// TwinCAT 3 PLC project IMD_PLC
// ProgramVersion: 3.1.4020.4
// libraries:
//   Tc2_ControllerToolbox, * (Beckhoff Automation GmbH)
//   Tc2_Database, * (Beckhoff Automation GmbH)
//   Tc2_Drive, * (Beckhoff Automation GmbH)
//   Tc2_EtherCAT, * (Beckhoff Automation GmbH)
//   Tc2_MC2, * (Beckhoff Automation GmbH)
//   Tc2_Standard, * (Beckhoff Automation GmbH)
//   Tc2_System, * (Beckhoff Automation GmbH)
//   Tc2_Utilities, * (Beckhoff Automation GmbH)
//   Tc3_Database, * (Beckhoff Automation GmbH)
//   Tc3_EventLogger, * (Beckhoff Automation GmbH)
//   Tc3_Module, * (Beckhoff Automation GmbH)
// project tree:
//   DUTs/ ST_COM_SpeedControl.TcDUT, ST_COM_IMD_SpdCntrl.TcDUT, ST_MachPar.TcDUT, ST_OEE.TcDUT, ST_PowerMeasurement.TcDUT, ST_ProdPar.TcDUT, ST_COM_SpdCntrl_IMD.TcDUT, ST_Record.TcDUT, ST_SysPar.TcDUT
//   GVLs/ GVL.TcGVL
//   / PlcTask.TcTTO, RecipeManager.TcRMO (not stored)
//   POUs/ FB_instancePath.TcPOU, HMI.TcPOU, MAIN.TcPOU, ST_Errors.TcDUT
//   POUs/InMoldDrying/BottomMold/ FB_BottomMold.TcPOU, ST_BottomMoldErrors.TcDUT, ST_BottomMoldMachPar.TcDUT, ST_BottomMoldProdPar.TcDUT, ST_BottomMoldSysPar.TcDUT
//   POUs/InMoldDrying/ FB_InMoldDrying.TcPOU, ST_IMDErrors.TcDUT, ST_IMDMachPar.TcDUT, ST_IMDProdPar.TcDUT, ST_IMDSysPar.TcDUT
//   POUs/InMoldDrying/HydrolicsMain/ FB_HydraulicsMain.TcPOU, ST_HydraulicsMainErrors.TcDUT, ST_HydraulicsMainMachPar.TcDUT
//   POUs/InMoldDrying/ProductForming/ FB_ProductForming.TcPOU, ST_FormingMoldErrors.TcDUT, ST_FormingMoldMachPar.TcDUT, ST_MachinePondErrors.TcDUT, ST_MachinePondMachPar.TcDUT, ST_ProductFormingErrors.TcDUT, ST_ProductFormingMachPar.TcDUT, ST_ProductFormingSysPar.TcDUT, ST_SpraybarErrors.TcDUT, ST_SpraybarMachPar.TcDUT
//   POUs/InMoldDrying/TopMold/ FB_TopMold.TcPOU, ST_TopMoldErrors.TcDUT, ST_TopMoldMachPar.TcDUT, ST_TopMoldProdPar.TcDUT
//   POUs/InMoldDrying/TransferMold/ FB_TransferMold.TcPOU, ST_TransferMoldErrors.TcDUT, ST_TransferMoldMachPar.TcDUT, ST_TransferMoldProdPar.TcDUT
//   POUs/ProductHandling/ FB_Gantry.TcPOU, FB_ProductHandling.TcPOU, ST_BlowOffProdPar.TcDUT, ST_GantryMachPar.TcDUT, ST_GantryProdPar.TcDUT, ST_GantryErrors.TcDUT, ST_GantrySysPar.TcDUT, ST_ProductHandlingErrors.TcDUT, ST_ProductHandlingMachPar.TcDUT, ST_ProductHandlingProdPar.TcDUT, ST_ProductHandlingSysPar.TcDUT
//   POUs/Standard/Analog/ FB_AnalogIn4_20mA.TcPOU, FB_AnalogInPT100.TcPOU, FB_AnalogOut0_10V.TcPOU, FB_AnalogOutMinus10_10V.TcPOU
//   POUs/Standard/Balluff/ FB_BalluffDevice.TcPOU, FB_BalluffPosition.TcPOU, ST_BalluffDevice.TcDUT, ST_BalluffMagnet.TcDUT
//   POUs/Standard/ FB_Blink.TcPOU, FB_EthercatDiag.TcPOU, GateRequest.TcPOU, UnixTimestamp.TcPOU
//   POUs/Standard/FIFO/ FB_CalculateMaxKO.TcPOU
//   POUs/Standard/HeatingZone/ FB_HeatingZone.TcPOU, ST_HeatingZoneErrors.TcDUT, ST_HeatingZone.TcDUT
//   POUs/Standard/HeatingZone/PID/ FB_1stOrderFilter.TcPOU, FB_PID.TcPOU, FB_PIDCtrl.TcPOU, FB_PID_CP.TcPOU, FB_PID_ROC.TcPOU, ST_PIDSettings.TcDUT
//   POUs/Standard/HydraulicCylinderAnalog/ FB_HydraulicCilinderAnalog.TcPOU, FB_HydraulicCilinderAnalog_.TcPOU, ST_HydraulicCilinderMachParAnalog.TcDUT, ST_HydraulicErrorsAnalog.TcDUT
//   POUs/Standard/Motor/ FB_Motor.TcPOU, FB_MotorSS.TcPOU, ST_MotorSSErrors.TcDUT, ST_MotorErrors.TcDUT
//   POUs/Standard/NC_Axis/ FB_NcAxis.TcPOU, ST_NcAxis_Errors.TcDUT, ST_NcAxis_Parameters_XX.TcDUT, ST_NcAxis_SysPar.TcDUT
//   POUs/Standard/HydraulicCilinder/ FB_HydraulicCilinder.TcPOU, ST_HydraulicCilinderMachPar.TcDUT, ST_HydraulicErrors.TcDUT
//   POUs/Standard/Valves/ FB_MonoValve2Fdbck.TcPOU, FB_CheckCilinder.TcPOU, FB_MonoValveNoFdbck.TcPOU, FB_BiValve2Fdbck.TcPOU, ST_CilinderErrors.TcDUT, ST_CilinderParameters.TcDUT
// real-time tasks:
//   TASK PlcTask: cycle T#10ms, priority 20, ADS port 350
//   TASK PlcTask_SpeedControl: cycle T#2ms, priority 19, ADS port 351
// motion (NC):
//   TASK NC-Task 1 SAF: cycle T#2ms, priority 4, ADS port 501
//   TASK NC-Task 1 SVB: cycle T#10ms, priority 8, ADS port 511
//   AXIS GantryA_Hor (id 1)
//     Dynamic: AccelerationMaximum=1657, DecelerationMaximum=1800, Acceleration=6750, Deceleration=6750, Jerk=50625
//     Velo: RefSearch=180, RefSync=180, SlowManual=165, FastManual=360, Fast=18000, Maximum=1800
//     OtherSettings: AllowMotionCmdToSlave=true
//     encoder EncType=8
//       EncPara: ScaleFactorNumerator=3.1607491629e-05, MaxCount=#xffffffff
//     drive DrvType=9
//       DrvPara: MaxCount=#xffffffff, DriveControlDWord=#x00030100
//         Analog: VeloReferenz=1657, VeloScale=1.02400649589962
//         TimeComp: TaskDelayCycles=1
//     controller CtrType=1
//       CtrPara: PriorControlFactor=1
//         PosDiffControl: Range=1
//         Observer: BandWidth=20
//   AXIS GantryA_Ver (id 2)
//     Dynamic: AccelerationMaximum=1000, DecelerationMaximum=1000, Acceleration=1000, Deceleration=1000, Jerk=15000
//     Velo: SlowManual=180, FastManual=450, Maximum=1000
//     OtherSettings: AllowMotionCmdToSlave=true
//     encoder EncType=8
//       EncPara: ScaleFactorNumerator=1.1444091797e-05, MaxCount=#xffffffff
//     drive DrvType=9
//       DrvPara: MaxCount=#xffffffff, DriveControlDWord=#x00030100
//         Analog: VeloReferenz=900, VeloScale=1.02400649589962
//         TimeComp: TaskDelayCycles=1
//     controller CtrType=1
//       CtrPara: PriorControlFactor=1
//         PosDiffControl: Range=0.3
//         Observer: BandWidth=20
//   AXIS GantryB_Hor (id 3)
//     Dynamic: Acceleration=5400, Deceleration=5400, Jerk=32400
//     Velo: SlowManual=165, FastManual=900, Maximum=1800
//     OtherSettings: AllowMotionCmdToSlave=true
//     encoder EncType=8
//       EncPara: ScaleFactorNumerator=3.1607491629e-05, Inverse=true, MaxCount=#xffffffff
//     drive DrvType=9
//       DrvPara: Inverse=true, MaxCount=#xffffffff, DriveControlDWord=#x00030100
//         Analog: VeloReferenz=1657, VeloScale=1.02400649589962
//         TimeComp: TaskDelayCycles=1
//     controller CtrType=1
//       CtrPara: PriorControlFactor=1
//         PosDiffControl: Range=1
//         Observer: BandWidth=20
//   AXIS GantryB_Ver (id 4)
//     Dynamic: Acceleration=3000, Deceleration=3000, Jerk=18000
//     Velo: FastManual=500, Maximum=1000
//     OtherSettings: AllowMotionCmdToSlave=true
//     encoder EncType=8
//       EncPara: ScaleFactorNumerator=1.1444091797e-05, Inverse=true, MaxCount=#xffffffff
//     drive DrvType=9
//       DrvPara: Inverse=true, MaxCount=#xffffffff, DriveControlDWord=#x00030100
//         Analog: VeloReferenz=900, VeloScale=1.02400649589962
//         TimeComp: TaskDelayCycles=1
//     controller CtrType=1
//       CtrPara: PriorControlFactor=1
//         PosDiffControl: Range=0.3
//         Observer: BandWidth=20
//   AXIS Conveyor (id 5)
//     General: UnitFlags=#x00000004
//     Dynamic: Acceleration=1368, Deceleration=1368, Jerk=8208
//     Velo: SlowManual=40, FastManual=207, Maximum=456
//     OtherSettings: AllowMotionCmdToSlave=true
//     encoder EncType=8
//       EncPara: ScaleFactorNumerator=7.780808382e-06, ModuloFactor=4620, Inverse=true, MaxCount=#xffffffff
//     drive DrvType=9
//       DrvPara: Inverse=true, MaxCount=#xffffffff, DriveControlDWord=#x00030100
//         Analog: VeloReferenz=414.74, VeloScale=1.02400649589962
//         TimeComp: TaskDelayCycles=1
//     controller CtrType=1
//       CtrPara: PriorControlFactor=1
//         Observer: BandWidth=20
//   AXIS SprayBar (id 6)
//     Dynamic: Acceleration=9780, Deceleration=9780, Jerk=58680
//     Velo: Maximum=3260
//     OtherSettings: AllowMotionCmdToSlave=true
//     encoder EncType=8
//       EncPara: ScaleFactorNumerator=5.8372727731e-05, MaxCount=#xffffffff
//     drive DrvType=9
//       DrvPara: MaxCount=#xffffffff, DriveControlDWord=#x00030100
//         Analog: VeloReferenz=2964, VeloScale=1.02400649589962
//         TimeComp: TaskDelayCycles=1
//     controller CtrType=1
//       CtrPara: PriorControlFactor=1
//         Observer: BandWidth=20
//   AXIS BottomMoldA (id 7)
//     Dynamic: AccelerationMaximum=5000, DecelerationMaximum=5000, Acceleration=1000, Deceleration=1000, Jerk=14000
//     Velo: Maximum=1250
//     OtherSettings: AllowMotionCmdToSlave=true
//     encoder EncType=8
//       EncPara: MaxCount=#xffffffff
//     drive DrvType=9
//       DrvPara: MaxCount=#xffffffff, DriveControlDWord=#x00030000
//         Analog: VeloScale=6
//         TimeComp: TaskDelayCycles=1
//     controller CtrType=1
//       CtrPara: PriorControlFactor=1
//         PosDiffControl: Enable=false, Range=15, Time=0
//         Observer: BandWidth=20
//   AXIS BottomMoldB (id 8)
//     Dynamic: Acceleration=1000, Deceleration=1000, Jerk=14000
//     OtherSettings: AllowMotionCmdToSlave=true
//     encoder EncType=8
//       EncPara: MaxCount=#xffffffff
//     drive DrvType=9
//       DrvPara: MaxCount=#xffffffff, DriveControlDWord=#x00030000
//         Analog: VeloScale=6
//         TimeComp: TaskDelayCycles=1
//     controller CtrType=1
//       CtrPara: PriorControlFactor=1
//         PosDiffControl: Enable=false
//         Observer: BandWidth=20
// I/O:
//   DEVICE Device 2 (EtherCAT) (disabled), AmsNetId 192.168.0.122.3.1
//     MCC01_600A1 (EK1100) [EK1100 EtherCAT Coupler (2A E-Bus)]
//       600A3 (EL9210) [EL9210 Power Supplier with LED (24V, Fuse, Diagnostics)]
//       600A4_TwinsafeController (EL6900) [EL6900, TwinSAFE PLC]
//       600A5 (EL2904) [EL2904, 4 Ch. Safety Output 24V, 0.5A, TwinSAFE]
//         modules: Module 1 (FSOES), Module 2 (DO)
//       600A6 (EL2904) [EL2904, 4 Ch. Safety Output 24V, 0.5A, TwinSAFE]
//         modules: Module 1 (FSOES), Module 2 (DO)
//       600A7 (EL2904) [EL2904, 4 Ch. Safety Output 24V, 0.5A, TwinSAFE]
//         modules: Module 1 (FSOES), Module 2 (DO)
//       600A8 (EL2904) [EL2904, 4 Ch. Safety Output 24V, 0.5A, TwinSAFE]
//         modules: Module 1 (FSOES), Module 2 (DO)
//       600A9 (EL9410) [EL9410 E-Bus Power Supplier  (Diagnostics)]
//       600A10 (EL2904) [EL2904, 4 Ch. Safety Output 24V, 0.5A, TwinSAFE]
//         modules: Module 1 (FSOES), Module 2 (DO)
//       600A11 (EL2904) [EL2904, 4 Ch. Safety Output 24V, 0.5A, TwinSAFE]
//         modules: Module 1 (FSOES), Module 2 (DO)
//       600A12 (EL2904) [EL2904, 4 Ch. Safety Output 24V, 0.5A, TwinSAFE]
//         modules: Module 1 (FSOES), Module 2 (DO)
//       600A13 (EL2904) [EL2904, 4 Ch. Safety Output 24V, 0.5A, TwinSAFE]
//         modules: Module 1 (FSOES), Module 2 (DO)
//       600A14 (EL2904) [EL2904, 4 Ch. Safety Output 24V, 0.5A, TwinSAFE]
//         modules: Module 1 (FSOES), Module 2 (DO)
//       600A15 (EL9210) [EL9210 Power Supplier with LED (24V, Fuse, Diagnostics)]
//       600A16 (EL1809) [EL1809 16Ch. Dig. Input 24V, 3ms]
//       600A17 (EL1809) [EL1809 16Ch. Dig. Input 24V, 3ms]
//       600A18 (EL1809) [EL1809 16Ch. Dig. Input 24V, 3ms]
//       600A19 (EL1809) [EL1809 16Ch. Dig. Input 24V, 3ms]
//       600A20 (EL1809) [EL1809 16Ch. Dig. Input 24V, 3ms]
//       600A21 (EL1809) [EL1809 16Ch. Dig. Input 24V, 3ms]
//       600A22 (EL9410) [EL9410 E-Bus Power Supplier  (Diagnostics)]
//       600A23 (EL2809) [EL2809 16Ch. Dig. Output 24V, 0.5A]
//       600A24 (EL2809) [EL2809 16Ch. Dig. Output 24V, 0.5A]
//       600A25 (EL2809) [EL2809 16Ch. Dig. Output 24V, 0.5A]
//       600A26 (EL2809) [EL2809 16Ch. Dig. Output 24V, 0.5A]
//       600A27 (EL2809) [EL2809 16Ch. Dig. Output 24V, 0.5A]
//       600A28 (EL9011) [EL9011 End Terminal]
//     MCC01_2_610A1 (EK1100) [EK1100 EtherCAT Coupler (2A E-Bus)]
//       610A1.1 (EL1809) [EL1809 16Ch. Dig. Input 24V, 3ms]
//       610A1.2 (EL2809) [EL2809 16Ch. Dig. Output 24V, 0.5A]
//       610A2 (EK1122) [EK1122 2 port EtherCAT junction]
//         Drive Gantry A (AX5203-0000-0203) [AX5203-0000-0203 EtherCAT Drive (SoE, 2 Ch.)]
//           GantryA (AX5805) [AX5805 (Safety Drive Option)]
//             modules: Module 1 (Safety Process Data, 2 axis), Module 2 (Standard Process Data, 2 axis)
//           Term 145 (EL9011) [EL9011 End Terminal]
//         Drive Gantry B (AX5203-0000-0203) [AX5203-0000-0203 EtherCAT Drive (SoE, 2 Ch.)]
//           GantryB (AX5805) [AX5805 (Safety Drive Option)]
//             modules: Module 1 (Safety Process Data, 2 axis), Module 2 (Standard Process Data, 2 axis)
//           Term 146 (EL9011) [EL9011 End Terminal]
//         Drive A-Belt / B-Spraybar (AX5201-0000-0203) [AX5201-0000-0203 EtherCAT Drive (SoE, 2 Ch.)]
//           SprayBar_Belt (AX5805) [AX5805 (Safety Drive Option)]
//             modules: Module 1 (Safety Process Data, 2 axis), Module 2 (Standard Process Data, 2 axis)
//           Term 147 (EL9011) [EL9011 End Terminal]
//         EJBox (EP9128-0021) [EP9128-0021 8x EtherCAT junction]
//           RIO_600A1 (EK1100) [EK1100 EtherCAT Coupler (2A E-Bus)]
//             RIO_600A2 (EL1804) [EL1804 4Ch. Dig. Input 24V, 3ms]
//             RIO_600A3 (EL1804) [EL1804 4Ch. Dig. Input 24V, 3ms]
//             RIO_600A4 (EL1804) [EL1804 4Ch. Dig. Input 24V, 3ms]
//             RIO_600A5 (EL1804) [EL1804 4Ch. Dig. Input 24V, 3ms]
//             RIO_600A6 (EL9210) [EL9210 Power Supplier with LED (24V, Fuse, Diagnostics)]
//             RIO_600A7 (EL2808) [EL2808 8Ch. Dig. Output 24V, 0.5A]
//             RIO_600A8 (EL2808) [EL2808 8Ch. Dig. Output 24V, 0.5A]
//             RIO_600A9 (EL2808) [EL2808 8Ch. Dig. Output 24V, 0.5A]
//             RIO_600A10 (EL9210) [EL9210 Power Supplier with LED (24V, Fuse, Diagnostics)]
//             RIO_600A11 (EL1904) [EL1904, 4 Ch. Safety Input 24V, TwinSAFE]
//               modules: Module 1 (FSOES)
//             RIO_600A12 (EL1904) [EL1904, 4 Ch. Safety Input 24V, TwinSAFE]
//               modules: Module 1 (FSOES)
//             RIO_600A13 (EL1904) [EL1904, 4 Ch. Safety Input 24V, TwinSAFE]
//               modules: Module 1 (FSOES)
//             RIO_600A14 (EL9410) [EL9410 E-Bus Power Supplier  (Diagnostics)]
//             RIO_600A15 (EL9210) [EL9210 Power Supplier with LED (24V, Fuse, Diagnostics)]
//             RIO_600A16 (EL1904) [EL1904, 4 Ch. Safety Input 24V, TwinSAFE]
//               modules: Module 1 (FSOES)
//             RIO_600A17 (EL1904) [EL1904, 4 Ch. Safety Input 24V, TwinSAFE]
//               modules: Module 1 (FSOES)
//             RIO_600A18 (EL9185) [EL9185 Potential Connection, 4 x 24-230V]
//             RIO_600A19 (EL9185) [EL9185 Potential Connection, 4 x 24-230V]
//             RIO_600A20 (EL1904) [EL1904, 4 Ch. Safety Input 24V, TwinSAFE]
//               modules: Module 1 (FSOES)
//             RIO_600A21 (EL1904) [EL1904, 4 Ch. Safety Input 24V, TwinSAFE]
//               modules: Module 1 (FSOES)
//             RIO_600A22 (EL1904) [EL1904, 4 Ch. Safety Input 24V, TwinSAFE]
//               modules: Module 1 (FSOES)
//             RIO_600A23 (EL1904) [EL1904, 4 Ch. Safety Input 24V, TwinSAFE]
//               modules: Module 1 (FSOES)
//             RIO_600A24 (EL1904) [EL1904, 4 Ch. Safety Input 24V, TwinSAFE]
//               modules: Module 1 (FSOES)
//             RIO_600A25 (EL1904) [EL1904, 4 Ch. Safety Input 24V, TwinSAFE]
//               modules: Module 1 (FSOES)
//             RIO_600A26 (EL1904) [EL1904, 4 Ch. Safety Input 24V, TwinSAFE]
//               modules: Module 1 (FSOES)
//             RIO_600A27 (EL9185) [EL9185 Potential Connection, 4 x 24-230V]
//             RIO_600A28 (EL9185) [EL9185 Potential Connection, 4 x 24-230V]
//             RIO_600A29 (EL9185) [EL9185 Potential Connection, 4 x 24-230V]
//             RIO_600A30 (EL9185) [EL9185 Potential Connection, 4 x 24-230V]
//             RIO_600A31 (EL3052) [EL3052 2Ch. Ana. Input 4-20mA]
//             RIO_600A32 (EL9011) [EL9011 End Terminal]
//           EPP_SensorSpeedControl (EPP1322-0001) [EPP1322-0001 3 port EtherCAT P gateway]
//             Box SpeedControl (EPP6228-0022) [EPP6228 (IO Link Master)]
//               modules: Module 1 (DeviceState Inputs Device), Module 2 (DeviceState Inputs), Module 3 (IO-Link Slave), Module 4 (empty), Module 5 (empty), Module 6 (empty), Module 7 (empty), Module 8 (empty), Module 9 (empty), Module 10 (empty), Module 11 (Digital Inputs)
//           TopMoldA (BTL7 EtherCAT) [BTL7 EtherCAT Modular]
//             modules: Module 1 (Position, speed, state, CAM and workarea), Module 17 (Error register and temperature), Module 18 (1 Magnet)
//           TransferMold (BTL7 EtherCAT) [BTL7 EtherCAT Modular]
//             modules: Module 1 (Position, speed, state, CAM and workarea), Module 17 (Error register and temperature), Module 18 (1 Magnet)
//           TopMoldB (BTL7 EtherCAT) [BTL7 EtherCAT Modular]
//             modules: Module 1 (Position, speed, state, CAM and workarea), Module 17 (Error register and temperature), Module 18 (1 Magnet)
//           BottomMoldHorizontal (BTL7 EtherCAT) [BTL7 EtherCAT Modular]
//             modules: Module 1 (Position, speed, state, CAM and workarea), Module 2 (Position, speed, state, CAM and workarea), Module 17 (Error register and temperature), Module 18 (2 Magnets)
//           MachinePond (BTL7 EtherCAT) [BTL7 EtherCAT Modular]
//             modules: Module 1 (Position, speed, state, CAM and workarea), Module 17 (Error register and temperature), Module 18 (1 Magnet)
//           JB_ (EP9128-1021) [EP9128-1021 8x EtherCAT junction - Dev A]
//             Box B (EP2008-0001) [EP2008-0001 8 Ch. Dig. Output 24V, 0,5A, M8]
//             Box Y1 [EP3174-0002 4Ch. Ana. Input +/-10V, 0-10V, 0/4-20mA configurable]
//             Box Y2 (EP3174-0002) [EP3174-0002 4Ch. Ana. Input +/-10V, 0-10V, 0/4-20mA configurable]
//             Box D (EP2028-0001) [EP2028-0001 8 Ch. Dig. Output 24V, 2A, M8]
//             Box A (EP2028-0001) [EP2028-0001 8 Ch. Dig. Output 24V, 2A, M8]
//             Box X (EP3174-0002) [EP3174-0002 4Ch. Ana. Input +/-10V, 0-10V, 0/4-20mA configurable]
//             Box C (EP2008-0001) [EP2008-0001 8 Ch. Dig. Output 24V, 0,5A, M8]
//             Box J (EP2008-0001) [EP2008-0001 8 Ch. Dig. Output 24V, 0,5A, M8]
//             Box AA (EP1008-0001) [EP1008-0001 8 Ch. Dig. Input 24V, 3ms, M8]
//             Box EF (EP2308-0001) [EP2308-0001 4 Ch. Dig. In, 3ms, 4 Ch. Dig. Out 24V, 0,5A, M8]
//             Box K (EP2008-0001) [EP2008-0001 8 Ch. Dig. Output 24V, 0,5A, M8]
//             Box L (EP1008-0001) [EP1008-0001 8 Ch. Dig. Input 24V, 3ms, M8]
//           JB_BottomMoldB_GantryA (EP9128-2021) [EP9128-2021 8x EtherCAT junction - Dev B]
//             Box HI (EP2308-0001) [EP2308-0001 4 Ch. Dig. In, 3ms, 4 Ch. Dig. Out 24V, 0,5A, M8]
//             Box M (EP2008-0001) [EP2008-0001 8 Ch. Dig. Output 24V, 0,5A, M8]
//             Box N (EP1008-0001) [EP1008-0001 8 Ch. Dig. Input 24V, 3ms, M8]
//             Box O (EP1008-0001) [EP1008-0001 8 Ch. Dig. Input 24V, 3ms, M8]
//             Box P (EP1008-0001) [EP1008-0001 8 Ch. Dig. Input 24V, 3ms, M8]
//             Box R (EP1008-0001) [EP1008-0001 8 Ch. Dig. Input 24V, 3ms, M8]
//             Box Q1 (EP2008-0001) [EP2008-0001 8 Ch. Dig. Output 24V, 0,5A, M8]
//             Box Q2 (EP2008-0001) [EP2008-0001 8 Ch. Dig. Output 24V, 0,5A, M8]
//         Box S (gantry B) (EP1008-0001) [EP1008-0001 8 Ch. Dig. Input 24V, 3ms, M8]
//         Box T (gantry B) (EP1008-0001) [EP1008-0001 8 Ch. Dig. Input 24V, 3ms, M8]
//         Box V (gantry B) (EP1008-0001) [EP1008-0001 8 Ch. Dig. Input 24V, 3ms, M8]
//         Box U1 (gantry B) (EP2008-0001) [EP2008-0001 8 Ch. Dig. Output 24V, 0,5A, M8]
//         Box U2 (gantry B) (EP2008-0001) [EP2008-0001 8 Ch. Dig. Output 24V, 0,5A, M8]
//       610A3 (EL9210) [EL9210 Power Supplier with LED (24V, Fuse, Diagnostics)]
//       610A4 (EL3403) [EL3403 3Ch. Power Measuring]
//       610A5 (EL3202) [EL3202 2Ch. Ana. Input PT100 (RTD)]
//       610A6 (EL3202) [EL3202 2Ch. Ana. Input PT100 (RTD)]
//       610A7 (EL3202) [EL3202 2Ch. Ana. Input PT100 (RTD)]
//       610A8 (EL3202) [EL3202 2Ch. Ana. Input PT100 (RTD)]
//       610A9 (EL3202) [EL3202 2Ch. Ana. Input PT100 (RTD)]
//       610A10 (EL3202) [EL3202 2Ch. Ana. Input PT100 (RTD)]
//       610A11 (EL3202) [EL3202 2Ch. Ana. Input PT100 (RTD)]
//       610A12 (EL9410) [EL9410 E-Bus Power Supplier  (Diagnostics)]
//       610A13 (EL3202) [EL3202 2Ch. Ana. Input PT100 (RTD)]
//       610A14 (EL3202) [EL3202 2Ch. Ana. Input PT100 (RTD)]
//       610A15 (EL3202) [EL3202 2Ch. Ana. Input PT100 (RTD)]
//       610A16 (EL3202) [EL3202 2Ch. Ana. Input PT100 (RTD)]
//       610A17 (EL3202) [EL3202 2Ch. Ana. Input PT100 (RTD)]
//       610A18 (EL9210) [EL9210 Power Supplier with LED (24V, Fuse, Diagnostics)]
//       610A19 (EL4002) [EL4002 2Ch. Ana. Output 0-10V, 12bit]
//       610A19.1 (EL3022) [EL3022 2Ch. Ana. Input 4-20mA DIFF]
//       610A20 (EL1904) [EL1904, 4 Ch. Safety Input 24V, TwinSAFE]
//         modules: Module 1 (FSOES)
//       610A21 (EL1904) [EL1904, 4 Ch. Safety Input 24V, TwinSAFE]
//         modules: Module 1 (FSOES)
//       610A22 (EL9011) [EL9011 End Terminal]
//     MCC02_600A1 (EK1100) [EK1100 EtherCAT Coupler (2A E-Bus)]
//       MCC02_600A2 (EL1904) [EL1904, 4 Ch. Safety Input 24V, TwinSAFE]
//         modules: Module 1 (FSOES)
//       MCC02_600A3 (EL1904) [EL1904, 4 Ch. Safety Input 24V, TwinSAFE]
//         modules: Module 1 (FSOES)
//       MCC02_600A4 (EL2904) [EL2904, 4 Ch. Safety Output 24V, 0.5A, TwinSAFE]
//         modules: Module 1 (FSOES), Module 2 (DO)
//       MCC02_600A5 (EL1809) [EL1809 16Ch. Dig. Input 24V, 3ms]
//       MCC02_600A6 (EL1809) [EL1809 16Ch. Dig. Input 24V, 3ms]
//       MCC02_600A7 (EL1809) [EL1809 16Ch. Dig. Input 24V, 3ms]
//       MCC02_600A8 (EL2809) [EL2809 16Ch. Dig. Output 24V, 0.5A]
//       MCC02_600A9 (EL4134) [EL4134 4Ch. Ana. Output -10/+10V, 16bit]
//       MCC02_600A10 (EL9011) [EL9011 End Terminal]
//     BottomMoldA (IndraDrive MPB20/21) [IndraDrive MPB20/21]
//     BottomMoldB (IndraDrive MPB20/21) [IndraDrive MPB20/21]
// variable links:
//   Device 2 (EtherCAT) <-> Device 2 (EtherCAT)/MCC01_2_610A1 (EK1100)/610A2 (EK1122)/Drive A-Belt / B-Spraybar (AX5201-0000-0203)/SprayBar_Belt (AX5805)
//     MCC01_600A1 (EK1100)/600A4_TwinsafeController (EL6900)/ConnectionInputs/Message_215 TxPDO <-> Module 1 (Safety Process Data, 2 axis)/Outputs (Controlword)/FSOE
//   Device 2 (EtherCAT) <-> Device 2 (EtherCAT)/MCC01_2_610A1 (EK1100)/610A2 (EK1122)/Drive Gantry A (AX5203-0000-0203)/GantryA (AX5805)
//     MCC01_600A1 (EK1100)/600A4_TwinsafeController (EL6900)/ConnectionOutputs/Message_213 RxPDO <-> Module 1 (Safety Process Data, 2 axis)/Inputs (Statusword)/FSOE
//   Device 2 (EtherCAT) <-> Device 2 (EtherCAT)/MCC01_2_610A1 (EK1100)/610A2 (EK1122)/Drive Gantry B (AX5203-0000-0203)/GantryB (AX5805)
//     MCC01_600A1 (EK1100)/600A4_TwinsafeController (EL6900)/ConnectionInputs/Message_214 TxPDO <-> Module 1 (Safety Process Data, 2 axis)/Outputs (Controlword)/FSOE
//   Device 2 (EtherCAT) <-> Device 2 (EtherCAT)/MCC01_2_610A1 (EK1100)/610A2 (EK1122)/EJBox (EP9128-0021)/RIO_600A1 (EK1100)/RIO_600A11 (EL1904)
//     MCC01_600A1 (EK1100)/600A4_TwinsafeController (EL6900)/ConnectionOutputs/Message_128 RxPDO <-> Module 1 (FSOES)/TxPDO/FSOE
//   Device 2 (EtherCAT) <-> Device 2 (EtherCAT)/MCC01_2_610A1 (EK1100)/610A2 (EK1122)/EJBox (EP9128-0021)/RIO_600A1 (EK1100)/RIO_600A13 (EL1904)
//     MCC01_600A1 (EK1100)/600A4_TwinsafeController (EL6900)/ConnectionOutputs/Message_130 RxPDO <-> Module 1 (FSOES)/TxPDO/FSOE
//   Device 2 (EtherCAT) <-> Device 2 (EtherCAT)/MCC01_2_610A1 (EK1100)/610A2 (EK1122)/EJBox (EP9128-0021)/RIO_600A1 (EK1100)/RIO_600A17 (EL1904)
//     MCC01_600A1 (EK1100)/600A4_TwinsafeController (EL6900)/ConnectionOutputs/Message_132 RxPDO <-> Module 1 (FSOES)/TxPDO/FSOE
//   Device 2 (EtherCAT) <-> Device 2 (EtherCAT)/MCC01_2_610A1 (EK1100)/610A2 (EK1122)/EJBox (EP9128-0021)/RIO_600A1 (EK1100)/RIO_600A20 (EL1904)
//     MCC01_600A1 (EK1100)/600A4_TwinsafeController (EL6900)/ConnectionInputs/Message_133 TxPDO <-> Module 1 (FSOES)/RxPDO/FSOE
//   Device 2 (EtherCAT) <-> Device 2 (EtherCAT)/MCC01_2_610A1 (EK1100)/610A2 (EK1122)/EJBox (EP9128-0021)/RIO_600A1 (EK1100)/RIO_600A21 (EL1904)
//     MCC01_600A1 (EK1100)/600A4_TwinsafeController (EL6900)/ConnectionInputs/Message_134 TxPDO <-> Module 1 (FSOES)/RxPDO/FSOE
//     MCC01_600A1 (EK1100)/600A4_TwinsafeController (EL6900)/ConnectionOutputs/Message_134 RxPDO <-> Module 1 (FSOES)/TxPDO/FSOE
//   Device 2 (EtherCAT) <-> Device 2 (EtherCAT)/MCC01_2_610A1 (EK1100)/610A2 (EK1122)/EJBox (EP9128-0021)/RIO_600A1 (EK1100)/RIO_600A22 (EL1904)
//     MCC01_600A1 (EK1100)/600A4_TwinsafeController (EL6900)/ConnectionInputs/Message_135 TxPDO <-> Module 1 (FSOES)/RxPDO/FSOE
//   Device 2 (EtherCAT) <-> Device 2 (EtherCAT)/MCC01_2_610A1 (EK1100)/610A2 (EK1122)/EJBox (EP9128-0021)/RIO_600A1 (EK1100)/RIO_600A23 (EL1904)
//     MCC01_600A1 (EK1100)/600A4_TwinsafeController (EL6900)/ConnectionInputs/Message_136 TxPDO <-> Module 1 (FSOES)/RxPDO/FSOE
//   Device 2 (EtherCAT) <-> Device 2 (EtherCAT)/MCC01_2_610A1 (EK1100)/610A2 (EK1122)/EJBox (EP9128-0021)/RIO_600A1 (EK1100)/RIO_600A24 (EL1904)
//     MCC01_600A1 (EK1100)/600A4_TwinsafeController (EL6900)/ConnectionInputs/Message_137 TxPDO <-> Module 1 (FSOES)/RxPDO/FSOE
//   Device 2 (EtherCAT) <-> Device 2 (EtherCAT)/MCC01_2_610A1 (EK1100)/610A2 (EK1122)/EJBox (EP9128-0021)/RIO_600A1 (EK1100)/RIO_600A25 (EL1904)
//     MCC01_600A1 (EK1100)/600A4_TwinsafeController (EL6900)/ConnectionInputs/Message_138 TxPDO <-> Module 1 (FSOES)/RxPDO/FSOE
//   Device 2 (EtherCAT) <-> Device 2 (EtherCAT)/MCC01_2_610A1 (EK1100)/610A2 (EK1122)/EJBox (EP9128-0021)/RIO_600A1 (EK1100)/RIO_600A26 (EL1904)
//     MCC01_600A1 (EK1100)/600A4_TwinsafeController (EL6900)/ConnectionInputs/Message_139 TxPDO <-> Module 1 (FSOES)/RxPDO/FSOE
//   Device 2 (EtherCAT) <-> Device 2 (EtherCAT)/MCC01_2_610A1 (EK1100)/610A20 (EL1904)
//     MCC01_600A1 (EK1100)/600A4_TwinsafeController (EL6900)/ConnectionOutputs/Message_140 RxPDO <-> Module 1 (FSOES)/TxPDO/FSOE
//   Device 2 (EtherCAT) <-> Device 2 (EtherCAT)/MCC01_600A1 (EK1100)/600A10 (EL2904)
//     MCC01_600A1 (EK1100)/600A4_TwinsafeController (EL6900)/ConnectionOutputs/Message_120 RxPDO <-> Module 1 (FSOES)/TxPDO/FSOE
//   Device 2 (EtherCAT) <-> Device 2 (EtherCAT)/MCC01_600A1 (EK1100)/600A11 (EL2904)
//     MCC01_600A1 (EK1100)/600A4_TwinsafeController (EL6900)/ConnectionInputs/Message_121 TxPDO <-> Module 1 (FSOES)/RxPDO/FSOE
//   Device 2 (EtherCAT) <-> Device 2 (EtherCAT)/MCC01_600A1 (EK1100)/600A13 (EL2904)
//     MCC01_600A1 (EK1100)/600A4_TwinsafeController (EL6900)/ConnectionInputs/Message_123 TxPDO <-> Module 1 (FSOES)/RxPDO/FSOE
//     MCC01_600A1 (EK1100)/600A4_TwinsafeController (EL6900)/ConnectionOutputs/Message_123 RxPDO <-> Module 1 (FSOES)/TxPDO/FSOE
//   Device 2 (EtherCAT) <-> Device 2 (EtherCAT)/MCC01_600A1 (EK1100)/600A16 (EL1809)
//     MCC01_600A1 (EK1100)/600A4_TwinsafeController (EL6900)/StandardOutputs/Standard In Var 142 <-> Channel 2/HydroPumpFB
//     MCC01_600A1 (EK1100)/600A4_TwinsafeController (EL6900)/StandardOutputs/Standard In Var 143 <-> Channel 5/PulpPumpFB
//   Device 2 (EtherCAT) <-> Device 2 (EtherCAT)/MCC01_600A1 (EK1100)/600A18 (EL1809)
//     MCC01_600A1 (EK1100)/600A4_TwinsafeController (EL6900)/StandardOutputs/Standard In Var 196 <-> Channel 16/Input
//   Device 2 (EtherCAT) <-> Device 2 (EtherCAT)/MCC01_600A1 (EK1100)/600A21 (EL1809)
//     MCC01_600A1 (EK1100)/600A4_TwinsafeController (EL6900)/StandardOutputs/Standard In Var 189 <-> Channel 2/Chan2
//     MCC01_600A1 (EK1100)/600A4_TwinsafeController (EL6900)/StandardOutputs/Standard In Var 190 <-> Channel 1/Chan1
//     MCC01_600A1 (EK1100)/600A4_TwinsafeController (EL6900)/StandardOutputs/Standard In Var 191 <-> Channel 3/Chan3
//     MCC01_600A1 (EK1100)/600A4_TwinsafeController (EL6900)/StandardOutputs/Standard In Var 192 <-> Channel 5/Chan5
//   Device 2 (EtherCAT) <-> Device 2 (EtherCAT)/MCC01_600A1 (EK1100)/600A4_TwinsafeController (EL6900)
//     MCC01_2_610A1 (EK1100)/610A2 (EK1122)/Drive A-Belt / B-Spraybar (AX5201-0000-0203)/SprayBar_Belt (AX5805)/Module 1 (Safety Process Data, 2 axis)/Inputs (Statusword)/FSOE <-> ConnectionOutputs/Message_215 RxPDO
//     MCC01_2_610A1 (EK1100)/610A2 (EK1122)/Drive Gantry A (AX5203-0000-0203)/GantryA (AX5805)/Module 1 (Safety Process Data, 2 axis)/Outputs (Controlword)/FSOE <-> ConnectionInputs/Message_213 TxPDO
//     MCC01_2_610A1 (EK1100)/610A2 (EK1122)/Drive Gantry B (AX5203-0000-0203)/GantryB (AX5805)/Module 1 (Safety Process Data, 2 axis)/Inputs (Statusword)/FSOE <-> ConnectionOutputs/Message_214 RxPDO
//     MCC01_2_610A1 (EK1100)/610A2 (EK1122)/EJBox (EP9128-0021)/RIO_600A1 (EK1100)/RIO_600A11 (EL1904)/Module 1 (FSOES)/RxPDO/FSOE <-> ConnectionInputs/Message_128 TxPDO
//     MCC01_2_610A1 (EK1100)/610A2 (EK1122)/EJBox (EP9128-0021)/RIO_600A1 (EK1100)/RIO_600A12 (EL1904)/Module 1 (FSOES)/RxPDO/FSOE <-> ConnectionInputs/Message_129 TxPDO
//     MCC01_2_610A1 (EK1100)/610A2 (EK1122)/EJBox (EP9128-0021)/RIO_600A1 (EK1100)/RIO_600A13 (EL1904)/Module 1 (FSOES)/RxPDO/FSOE <-> ConnectionInputs/Message_130 TxPDO
//     MCC01_2_610A1 (EK1100)/610A2 (EK1122)/EJBox (EP9128-0021)/RIO_600A1 (EK1100)/RIO_600A16 (EL1904)/Module 1 (FSOES)/RxPDO/FSOE <-> ConnectionInputs/Message_131 TxPDO
//     MCC01_2_610A1 (EK1100)/610A2 (EK1122)/EJBox (EP9128-0021)/RIO_600A1 (EK1100)/RIO_600A17 (EL1904)/Module 1 (FSOES)/RxPDO/FSOE <-> ConnectionInputs/Message_132 TxPDO
//     MCC01_2_610A1 (EK1100)/610A2 (EK1122)/EJBox (EP9128-0021)/RIO_600A1 (EK1100)/RIO_600A12 (EL1904)/Module 1 (FSOES)/TxPDO/FSOE <-> ConnectionOutputs/Message_129 RxPDO
//     MCC01_2_610A1 (EK1100)/610A2 (EK1122)/EJBox (EP9128-0021)/RIO_600A1 (EK1100)/RIO_600A16 (EL1904)/Module 1 (FSOES)/TxPDO/FSOE <-> ConnectionOutputs/Message_131 RxPDO
//     MCC01_2_610A1 (EK1100)/610A2 (EK1122)/EJBox (EP9128-0021)/RIO_600A1 (EK1100)/RIO_600A20 (EL1904)/Module 1 (FSOES)/TxPDO/FSOE <-> ConnectionOutputs/Message_133 RxPDO
//     MCC01_2_610A1 (EK1100)/610A2 (EK1122)/EJBox (EP9128-0021)/RIO_600A1 (EK1100)/RIO_600A22 (EL1904)/Module 1 (FSOES)/TxPDO/FSOE <-> ConnectionOutputs/Message_135 RxPDO
//     MCC01_2_610A1 (EK1100)/610A2 (EK1122)/EJBox (EP9128-0021)/RIO_600A1 (EK1100)/RIO_600A23 (EL1904)/Module 1 (FSOES)/TxPDO/FSOE <-> ConnectionOutputs/Message_136 RxPDO
//     MCC01_2_610A1 (EK1100)/610A2 (EK1122)/EJBox (EP9128-0021)/RIO_600A1 (EK1100)/RIO_600A24 (EL1904)/Module 1 (FSOES)/TxPDO/FSOE <-> ConnectionOutputs/Message_137 RxPDO
//     MCC01_2_610A1 (EK1100)/610A2 (EK1122)/EJBox (EP9128-0021)/RIO_600A1 (EK1100)/RIO_600A25 (EL1904)/Module 1 (FSOES)/TxPDO/FSOE <-> ConnectionOutputs/Message_138 RxPDO
//     MCC01_2_610A1 (EK1100)/610A2 (EK1122)/EJBox (EP9128-0021)/RIO_600A1 (EK1100)/RIO_600A26 (EL1904)/Module 1 (FSOES)/TxPDO/FSOE <-> ConnectionOutputs/Message_139 RxPDO
//     MCC01_2_610A1 (EK1100)/610A20 (EL1904)/Module 1 (FSOES)/RxPDO/FSOE <-> ConnectionInputs/Message_140 TxPDO
//     MCC01_2_610A1 (EK1100)/610A21 (EL1904)/Module 1 (FSOES)/RxPDO/FSOE <-> ConnectionInputs/Message_141 TxPDO
//     MCC01_2_610A1 (EK1100)/610A21 (EL1904)/Module 1 (FSOES)/TxPDO/FSOE <-> ConnectionOutputs/Message_141 RxPDO
//     MCC01_600A1 (EK1100)/600A10 (EL2904)/Module 1 (FSOES)/RxPDO/FSOE <-> ConnectionInputs/Message_120 TxPDO
//     MCC01_600A1 (EK1100)/600A12 (EL2904)/Module 1 (FSOES)/RxPDO/FSOE <-> ConnectionInputs/Message_122 TxPDO
//     MCC01_600A1 (EK1100)/600A14 (EL2904)/Module 1 (FSOES)/RxPDO/FSOE <-> ConnectionInputs/Message_124 TxPDO
//     MCC01_600A1 (EK1100)/600A5 (EL2904)/Module 1 (FSOES)/RxPDO/FSOE <-> ConnectionInputs/Message_116 TxPDO
//     MCC01_600A1 (EK1100)/600A7 (EL2904)/Module 1 (FSOES)/RxPDO/FSOE <-> ConnectionInputs/Message_118 TxPDO
//     MCC01_600A1 (EK1100)/600A8 (EL2904)/Module 1 (FSOES)/RxPDO/FSOE <-> ConnectionInputs/Message_119 TxPDO
//     MCC01_600A1 (EK1100)/600A11 (EL2904)/Module 1 (FSOES)/TxPDO/FSOE <-> ConnectionOutputs/Message_121 RxPDO
//     MCC01_600A1 (EK1100)/600A12 (EL2904)/Module 1 (FSOES)/TxPDO/FSOE <-> ConnectionOutputs/Message_122 RxPDO
//     MCC01_600A1 (EK1100)/600A14 (EL2904)/Module 1 (FSOES)/TxPDO/FSOE <-> ConnectionOutputs/Message_124 RxPDO
//     MCC01_600A1 (EK1100)/600A21 (EL1809)/Channel 4/Chan4 <-> StandardOutputs/Standard In Var 188
//     MCC02_600A1 (EK1100)/MCC02_600A3 (EL1904)/Module 1 (FSOES)/RxPDO/FSOE <-> ConnectionInputs/Message_223 TxPDO
//     MCC02_600A1 (EK1100)/MCC02_600A4 (EL2904)/Module 1 (FSOES)/RxPDO/FSOE <-> ConnectionInputs/Message_218 TxPDO
//     MCC02_600A1 (EK1100)/MCC02_600A6 (EL1809)/Channel 13/Input <-> StandardOutputs/Standard In Var 220
//   Device 2 (EtherCAT) <-> Device 2 (EtherCAT)/MCC01_600A1 (EK1100)/600A5 (EL2904)
//     MCC01_600A1 (EK1100)/600A4_TwinsafeController (EL6900)/ConnectionOutputs/Message_116 RxPDO <-> Module 1 (FSOES)/TxPDO/FSOE
//   Device 2 (EtherCAT) <-> Device 2 (EtherCAT)/MCC01_600A1 (EK1100)/600A6 (EL2904)
//     MCC01_600A1 (EK1100)/600A4_TwinsafeController (EL6900)/ConnectionInputs/Message_117 TxPDO <-> Module 1 (FSOES)/RxPDO/FSOE
//     MCC01_600A1 (EK1100)/600A4_TwinsafeController (EL6900)/ConnectionOutputs/Message_117 RxPDO <-> Module 1 (FSOES)/TxPDO/FSOE
//   Device 2 (EtherCAT) <-> Device 2 (EtherCAT)/MCC01_600A1 (EK1100)/600A7 (EL2904)
//     MCC01_600A1 (EK1100)/600A4_TwinsafeController (EL6900)/ConnectionOutputs/Message_118 RxPDO <-> Module 1 (FSOES)/TxPDO/FSOE
//   Device 2 (EtherCAT) <-> Device 2 (EtherCAT)/MCC01_600A1 (EK1100)/600A8 (EL2904)
//     MCC01_600A1 (EK1100)/600A4_TwinsafeController (EL6900)/ConnectionOutputs/Message_119 RxPDO <-> Module 1 (FSOES)/TxPDO/FSOE
//   Device 2 (EtherCAT) <-> Device 2 (EtherCAT)/MCC02_600A1 (EK1100)/MCC02_600A2 (EL1904)
//     MCC01_600A1 (EK1100)/600A4_TwinsafeController (EL6900)/ConnectionInputs/Message_222 TxPDO <-> Module 1 (FSOES)/RxPDO/FSOE
//     MCC01_600A1 (EK1100)/600A4_TwinsafeController (EL6900)/ConnectionOutputs/Message_222 RxPDO <-> Module 1 (FSOES)/TxPDO/FSOE
//   Device 2 (EtherCAT) <-> Device 2 (EtherCAT)/MCC02_600A1 (EK1100)/MCC02_600A3 (EL1904)
//     MCC01_600A1 (EK1100)/600A4_TwinsafeController (EL6900)/ConnectionOutputs/Message_223 RxPDO <-> Module 1 (FSOES)/TxPDO/FSOE
//   Device 2 (EtherCAT) <-> Device 2 (EtherCAT)/MCC02_600A1 (EK1100)/MCC02_600A4 (EL2904)
//     MCC01_600A1 (EK1100)/600A4_TwinsafeController (EL6900)/ConnectionOutputs/Message_218 RxPDO <-> Module 1 (FSOES)/TxPDO/FSOE
//   Device 2 (EtherCAT) <-> Device 2 (EtherCAT)/MCC02_600A1 (EK1100)/MCC02_600A5 (EL1809)
//     MCC01_600A1 (EK1100)/600A4_TwinsafeController (EL6900)/StandardOutputs/Standard In Var 221 <-> Channel 5/Input
//   NC-Task 1 SAF/Axes/BottomMoldA <-> Device 2 (EtherCAT)/BottomMoldA (IndraDrive MPB20/21)
//     Drive/Inputs/In/nDcOutputTime <-> InfoData/DcOutputShift
//     Drive/Inputs/In/nState1 <-> AT/Drive status word @bit 8
//     Drive/Inputs/In/nState2 <-> AT/Drive status word
//     Drive/Inputs/In/nState4 @bit 1 <-> WcState/InputToggle
//     Drive/Inputs/In/nState4 <-> WcState/WcState
//     Drive/Outputs/Out/nCtrl1 <-> MDT/Master control word @bit 8
//     Drive/Outputs/Out/nDataOut1 <-> MDT/Position command value
//     Enc/Inputs/In/nDataIn1 <-> AT/Position feedback value 1
//     Enc/Inputs/In/nDcInputTime <-> InfoData/DcInputShift
//     Enc/Inputs/In/nState4 @bit 1 <-> WcState/InputToggle
//     Enc/Inputs/In/nState4 <-> WcState/WcState
//   NC-Task 1 SAF/Axes/BottomMoldB <-> Device 2 (EtherCAT)/BottomMoldB (IndraDrive MPB20/21)
//     Drive/Inputs/In/nDcOutputTime <-> InfoData/DcOutputShift
//     Drive/Inputs/In/nState1 <-> AT/Drive status word @bit 8
//     Drive/Inputs/In/nState2 <-> AT/Drive status word
//     Drive/Inputs/In/nState4 @bit 1 <-> WcState/InputToggle
//     Drive/Inputs/In/nState4 <-> WcState/WcState
//     Drive/Outputs/Out/nCtrl1 <-> MDT/Master control word @bit 8
//     Drive/Outputs/Out/nDataOut1 <-> MDT/Position command value
//     Enc/Inputs/In/nDataIn1 <-> AT/Position feedback value 1
//     Enc/Inputs/In/nDcInputTime <-> InfoData/DcInputShift
//     Enc/Inputs/In/nState4 @bit 1 <-> WcState/InputToggle
//     Enc/Inputs/In/nState4 <-> WcState/WcState
//   NC-Task 1 SAF/Axes/Conveyor <-> Device 2 (EtherCAT)/MCC01_2_610A1 (EK1100)/610A2 (EK1122)/Drive A-Belt / B-Spraybar (AX5201-0000-0203)
//     Drive/Inputs/In/nDataIn1 <-> AT 1/Following distance
//     Drive/Inputs/In/nDcOutputTime <-> InfoData/DcOutputShift
//     Drive/Inputs/In/nState1 <-> AT 1/Drive status word @bit 8
//     Drive/Inputs/In/nState2 <-> AT 1/Drive status word
//     Drive/Inputs/In/nState4 @bit 1 <-> WcState/InputToggle
//     Drive/Inputs/In/nState4 <-> WcState/WcState
//     Drive/Outputs/Out/nCtrl1 <-> MDT 1/Master control word @bit 8
//     Drive/Outputs/Out/nDataOut1 <-> MDT 1/Position command value
//     Enc/Inputs/In/nDataIn1 <-> AT 1/Position feedback 1 value
//     Enc/Inputs/In/nDcInputTime <-> InfoData/DcInputShift
//     Enc/Inputs/In/nState4 @bit 1 <-> WcState/InputToggle
//     Enc/Inputs/In/nState4 <-> WcState/WcState
//   NC-Task 1 SAF/Axes/GantryA_Hor <-> Device 2 (EtherCAT)/MCC01_2_610A1 (EK1100)/610A2 (EK1122)/Drive Gantry A (AX5203-0000-0203)
//     Drive/Inputs/In/nDataIn1 <-> AT 1/Following distance
//     Drive/Inputs/In/nDataIn3[0] <-> AT 1/Torque feedback value
//     Drive/Inputs/In/nDcOutputTime <-> InfoData/DcOutputShift
//     Drive/Inputs/In/nState1 <-> AT 1/Drive status word @bit 8
//     Drive/Inputs/In/nState2 <-> AT 1/Drive status word
//     Drive/Inputs/In/nState4 @bit 1 <-> WcState/InputToggle
//     Drive/Inputs/In/nState4 <-> WcState/WcState
//     Drive/Outputs/Out/nCtrl1 <-> MDT 1/Master control word @bit 8
//     Drive/Outputs/Out/nDataOut1 <-> MDT 1/Position command value
//     Enc/Inputs/In/nDataIn1 <-> AT 1/Position feedback 1 value
//     Enc/Inputs/In/nDcInputTime <-> InfoData/DcInputShift
//     Enc/Inputs/In/nState4 @bit 1 <-> WcState/InputToggle
//     Enc/Inputs/In/nState4 <-> WcState/WcState
//   NC-Task 1 SAF/Axes/GantryA_Ver <-> Device 2 (EtherCAT)/MCC01_2_610A1 (EK1100)/610A2 (EK1122)/Drive Gantry A (AX5203-0000-0203)
//     Drive/Inputs/In/nDataIn1 <-> AT 2/Following distance
//     Drive/Inputs/In/nDataIn3[0] <-> AT 2/Torque feedback value
//     Drive/Inputs/In/nDcOutputTime <-> InfoData/DcOutputShift
//     Drive/Inputs/In/nState1 <-> AT 2/Drive status word @bit 8
//     Drive/Inputs/In/nState2 <-> AT 2/Drive status word
//     Drive/Inputs/In/nState4 @bit 1 <-> WcState/InputToggle
//     Drive/Inputs/In/nState4 <-> WcState/WcState
//     Drive/Outputs/Out/nCtrl1 <-> MDT 2/Master control word @bit 8
//     Drive/Outputs/Out/nDataOut1 <-> MDT 2/Position command value
//     Enc/Inputs/In/nDataIn1 <-> AT 2/Position feedback 1 value
//     Enc/Inputs/In/nDcInputTime <-> InfoData/DcInputShift
//     Enc/Inputs/In/nState4 @bit 1 <-> WcState/InputToggle
//     Enc/Inputs/In/nState4 <-> WcState/WcState
//   NC-Task 1 SAF/Axes/GantryB_Hor <-> Device 2 (EtherCAT)/MCC01_2_610A1 (EK1100)/610A2 (EK1122)/Drive Gantry B (AX5203-0000-0203)
//     Drive/Inputs/In/nDataIn1 <-> AT 1/Following distance
//     Drive/Inputs/In/nDcOutputTime <-> InfoData/DcOutputShift
//     Drive/Inputs/In/nState1 <-> AT 1/Drive status word @bit 8
//     Drive/Inputs/In/nState2 <-> AT 1/Drive status word
//     Drive/Inputs/In/nState4 @bit 1 <-> WcState/InputToggle
//     Drive/Inputs/In/nState4 <-> WcState/WcState
//     Drive/Outputs/Out/nCtrl1 <-> MDT 1/Master control word @bit 8
//     Drive/Outputs/Out/nDataOut1 <-> MDT 1/Position command value
//     Enc/Inputs/In/nDataIn1 <-> AT 1/Position feedback 1 value
//     Enc/Inputs/In/nDcInputTime <-> InfoData/DcInputShift
//     Enc/Inputs/In/nState4 @bit 1 <-> WcState/InputToggle
//     Enc/Inputs/In/nState4 <-> WcState/WcState
//   NC-Task 1 SAF/Axes/GantryB_Ver <-> Device 2 (EtherCAT)/MCC01_2_610A1 (EK1100)/610A2 (EK1122)/Drive Gantry B (AX5203-0000-0203)
//     Drive/Inputs/In/nDataIn1 <-> AT 2/Following distance
//     Drive/Inputs/In/nDcOutputTime <-> InfoData/DcOutputShift
//     Drive/Inputs/In/nState1 <-> AT 2/Drive status word @bit 8
//     Drive/Inputs/In/nState2 <-> AT 2/Drive status word
//     Drive/Inputs/In/nState4 @bit 1 <-> WcState/InputToggle
//     Drive/Inputs/In/nState4 <-> WcState/WcState
//     Drive/Outputs/Out/nCtrl1 <-> MDT 2/Master control word @bit 8
//     Drive/Outputs/Out/nDataOut1 <-> MDT 2/Position command value
//     Enc/Inputs/In/nDataIn1 <-> AT 2/Position feedback 1 value
//     Enc/Inputs/In/nDcInputTime <-> InfoData/DcInputShift
//     Enc/Inputs/In/nState4 @bit 1 <-> WcState/InputToggle
//     Enc/Inputs/In/nState4 <-> WcState/WcState
//   NC-Task 1 SAF/Axes/SprayBar <-> Device 2 (EtherCAT)/MCC01_2_610A1 (EK1100)/610A2 (EK1122)/Drive A-Belt / B-Spraybar (AX5201-0000-0203)
//     Drive/Inputs/In/nDataIn1 <-> AT 2/Following distance
//     Drive/Inputs/In/nDcOutputTime <-> InfoData/DcOutputShift
//     Drive/Inputs/In/nState1 <-> AT 2/Drive status word @bit 8
//     Drive/Inputs/In/nState2 <-> AT 2/Drive status word
//     Drive/Inputs/In/nState4 @bit 1 <-> WcState/InputToggle
//     Drive/Inputs/In/nState4 <-> WcState/WcState
//     Drive/Outputs/Out/nCtrl1 <-> MDT 2/Master control word @bit 8
//     Drive/Outputs/Out/nDataOut1 <-> MDT 2/Position command value
//     Enc/Inputs/In/nDataIn1 <-> AT 2/Position feedback 1 value
//     Enc/Inputs/In/nDcInputTime <-> InfoData/DcInputShift
//     Enc/Inputs/In/nState4 @bit 1 <-> WcState/InputToggle
//     Enc/Inputs/In/nState4 <-> WcState/WcState
//   IMD_PLC/IMD_PLC Instance <-> Device 2 (EtherCAT)
//     PlcTask Inputs/MAIN.iAmsNetID <-> InfoData/AmsNetId
//     PlcTask Inputs/MAIN.iwCfgSlaveCount <-> InfoData/CfgSlaveCount
//     PlcTask Inputs/MAIN.iwDevID <-> InfoData/DevId
//     PlcTask Inputs/MAIN.iwDevState <-> Inputs/DevState
//     PlcTask Inputs/MAIN.iwSlaveCount <-> Inputs/SlaveCount
//   IMD_PLC/IMD_PLC Instance <-> Device 2 (EtherCAT)/BottomMoldA (IndraDrive MPB20/21)
//     PlcTask Inputs/MAIN.InMoldDrying.BottomMoldA.HorizontalAxis.iDriveRef/aNetId <-> InfoData/AdsAddr/netId
//     PlcTask Inputs/MAIN.InMoldDrying.BottomMoldA.HorizontalAxis.iDriveRef/nSlaveAddr <-> InfoData/AdsAddr/port
//   IMD_PLC/IMD_PLC Instance <-> Device 2 (EtherCAT)/BottomMoldB (IndraDrive MPB20/21)
//     PlcTask Inputs/MAIN.InMoldDrying.BottomMoldB.HorizontalAxis.iDriveRef/aNetId <-> InfoData/AdsAddr/netId
//     PlcTask Inputs/MAIN.InMoldDrying.BottomMoldB.HorizontalAxis.iDriveRef/nSlaveAddr <-> InfoData/AdsAddr/port
//   IMD_PLC/IMD_PLC Instance <-> Device 2 (EtherCAT)/MCC01_2_610A1 (EK1100)/610A1.1 (EL1809)
//     PlcTask Inputs/MAIN.ixMainSwitchOFF <-> Channel 1/Input
//     PlcTask Inputs/MAIN.ixUPS_Alarm <-> Channel 2/Input
//     PlcTask Inputs/MAIN.ixUPS_BatMode <-> Channel 3/Input
//     PlcTask Inputs/MAIN.ixUPS_Charge <-> Channel 4/Input
//   IMD_PLC/IMD_PLC Instance <-> Device 2 (EtherCAT)/MCC01_2_610A1 (EK1100)/610A1.2 (EL2809)
//     PlcTask Outputs/MAIN.qxPcRemoteOff <-> Channel 1/Output
//   IMD_PLC/IMD_PLC Instance <-> Device 2 (EtherCAT)/MCC01_2_610A1 (EK1100)/610A10 (EL3202)
//     PlcTask Inputs/MAIN.InMoldDrying.BottomMoldA.HeatingZone[5].FB_Temperature.RawInput <-> RTD Inputs Channel 1/Value
//     PlcTask Inputs/MAIN.InMoldDrying.BottomMoldA.HeatingZone[6].FB_Temperature.RawInput <-> RTD Inputs Channel 2/Value
//     PlcTask Inputs/MAIN.InMoldDrying.BottomMoldA.HeatingZone[5].FB_Temperature.Status <-> RTD Inputs Channel 1/Status
//     PlcTask Inputs/MAIN.InMoldDrying.BottomMoldA.HeatingZone[6].FB_Temperature.Status <-> RTD Inputs Channel 2/Status
//   IMD_PLC/IMD_PLC Instance <-> Device 2 (EtherCAT)/MCC01_2_610A1 (EK1100)/610A11 (EL3202)
//     PlcTask Inputs/MAIN.InMoldDrying.TopMoldB.HeatingZone[1].FB_Temperature.RawInput <-> RTD Inputs Channel 1/Value
//     PlcTask Inputs/MAIN.InMoldDrying.TopMoldB.HeatingZone[2].FB_Temperature.RawInput <-> RTD Inputs Channel 2/Value
//     PlcTask Inputs/MAIN.InMoldDrying.TopMoldB.HeatingZone[1].FB_Temperature.Status <-> RTD Inputs Channel 1/Status
//     PlcTask Inputs/MAIN.InMoldDrying.TopMoldB.HeatingZone[2].FB_Temperature.Status <-> RTD Inputs Channel 2/Status
//   IMD_PLC/IMD_PLC Instance <-> Device 2 (EtherCAT)/MCC01_2_610A1 (EK1100)/610A13 (EL3202)
//     PlcTask Inputs/MAIN.InMoldDrying.TopMoldB.HeatingZone[3].FB_Temperature.RawInput <-> RTD Inputs Channel 1/Value
//     PlcTask Inputs/MAIN.InMoldDrying.TopMoldB.HeatingZone[4].FB_Temperature.RawInput <-> RTD Inputs Channel 2/Value
//     PlcTask Inputs/MAIN.InMoldDrying.TopMoldB.HeatingZone[3].FB_Temperature.Status <-> RTD Inputs Channel 1/Status
//     PlcTask Inputs/MAIN.InMoldDrying.TopMoldB.HeatingZone[4].FB_Temperature.Status <-> RTD Inputs Channel 2/Status
//   IMD_PLC/IMD_PLC Instance <-> Device 2 (EtherCAT)/MCC01_2_610A1 (EK1100)/610A14 (EL3202)
//     PlcTask Inputs/MAIN.InMoldDrying.TopMoldB.HeatingZone[5].FB_Temperature.RawInput <-> RTD Inputs Channel 1/Value
//     PlcTask Inputs/MAIN.InMoldDrying.TopMoldB.HeatingZone[6].FB_Temperature.RawInput <-> RTD Inputs Channel 2/Value
//     PlcTask Inputs/MAIN.InMoldDrying.TopMoldB.HeatingZone[5].FB_Temperature.Status <-> RTD Inputs Channel 1/Status
//     PlcTask Inputs/MAIN.InMoldDrying.TopMoldB.HeatingZone[6].FB_Temperature.Status <-> RTD Inputs Channel 2/Status
//   IMD_PLC/IMD_PLC Instance <-> Device 2 (EtherCAT)/MCC01_2_610A1 (EK1100)/610A15 (EL3202)
//     PlcTask Inputs/MAIN.InMoldDrying.BottomMoldB.HeatingZone[1].FB_Temperature.RawInput <-> RTD Inputs Channel 1/Value
//     PlcTask Inputs/MAIN.InMoldDrying.BottomMoldB.HeatingZone[2].FB_Temperature.RawInput <-> RTD Inputs Channel 2/Value
//     PlcTask Inputs/MAIN.InMoldDrying.BottomMoldB.HeatingZone[1].FB_Temperature.Status <-> RTD Inputs Channel 1/Status
//     PlcTask Inputs/MAIN.InMoldDrying.BottomMoldB.HeatingZone[2].FB_Temperature.Status <-> RTD Inputs Channel 2/Status
//   IMD_PLC/IMD_PLC Instance <-> Device 2 (EtherCAT)/MCC01_2_610A1 (EK1100)/610A16 (EL3202)
//     PlcTask Inputs/MAIN.InMoldDrying.BottomMoldB.HeatingZone[3].FB_Temperature.RawInput <-> RTD Inputs Channel 1/Value
//     PlcTask Inputs/MAIN.InMoldDrying.BottomMoldB.HeatingZone[4].FB_Temperature.RawInput <-> RTD Inputs Channel 2/Value
//     PlcTask Inputs/MAIN.InMoldDrying.BottomMoldB.HeatingZone[3].FB_Temperature.Status <-> RTD Inputs Channel 1/Status
//     PlcTask Inputs/MAIN.InMoldDrying.BottomMoldB.HeatingZone[4].FB_Temperature.Status <-> RTD Inputs Channel 2/Status
//   IMD_PLC/IMD_PLC Instance <-> Device 2 (EtherCAT)/MCC01_2_610A1 (EK1100)/610A17 (EL3202)
//     PlcTask Inputs/MAIN.InMoldDrying.BottomMoldB.HeatingZone[5].FB_Temperature.RawInput <-> RTD Inputs Channel 1/Value
//     PlcTask Inputs/MAIN.InMoldDrying.BottomMoldB.HeatingZone[6].FB_Temperature.RawInput <-> RTD Inputs Channel 2/Value
//     PlcTask Inputs/MAIN.InMoldDrying.BottomMoldB.HeatingZone[5].FB_Temperature.Status <-> RTD Inputs Channel 1/Status
//     PlcTask Inputs/MAIN.InMoldDrying.BottomMoldB.HeatingZone[6].FB_Temperature.Status <-> RTD Inputs Channel 2/Status
//   IMD_PLC/IMD_PLC Instance <-> Device 2 (EtherCAT)/MCC01_2_610A1 (EK1100)/610A19.1 (EL3022)
//     PlcTask Inputs/MAIN.InMoldDrying.ProductForming.TankLevel01.RawInput <-> AI Standard Channel 1/Value
//     PlcTask Inputs/MAIN.InMoldDrying.ProductForming.TankLevel02.RawInput <-> AI Standard Channel 2/Value
//   IMD_PLC/IMD_PLC Instance <-> Device 2 (EtherCAT)/MCC01_2_610A1 (EK1100)/610A2 (EK1122)/Box S (gantry B) (EP1008-0001)
//     PlcTask Inputs/MAIN.ProductHandling.GantryB.ixEndLimitHorBack <-> Channel 2/Input
//     PlcTask Inputs/MAIN.ProductHandling.GantryB.ixEndLimitHorFront <-> Channel 1/Input
//   IMD_PLC/IMD_PLC Instance <-> Device 2 (EtherCAT)/MCC01_2_610A1 (EK1100)/610A2 (EK1122)/Box T (gantry B) (EP1008-0001)
//     PlcTask Inputs/MAIN.ProductHandling.GantryB.ixEndLimitVertDown <-> Channel 2/Input
//     PlcTask Inputs/MAIN.ProductHandling.GantryB.ixEndLimitVertUp <-> Channel 1/Input
//   IMD_PLC/IMD_PLC Instance <-> Device 2 (EtherCAT)/MCC01_2_610A1 (EK1100)/610A2 (EK1122)/Box U1 (gantry B) (EP2008-0001)
//     PlcTask Outputs/MAIN.ProductHandling.GantryB.BlowOff[{1..4}].Q <-> Channel {2..8 step 2}/Output  (4 links)
//     PlcTask Outputs/MAIN.ProductHandling.GantryB.VacuumValve[{1..4}].Q <-> Channel {1..7 step 2}/Output  (4 links)
//   IMD_PLC/IMD_PLC Instance <-> Device 2 (EtherCAT)/MCC01_2_610A1 (EK1100)/610A2 (EK1122)/Box U2 (gantry B) (EP2008-0001)
//     PlcTask Outputs/MAIN.ProductHandling.GantryB.BlowOff[5].Q <-> Channel 2/Output
//     PlcTask Outputs/MAIN.ProductHandling.GantryB.VacuumValve[5].Q <-> Channel 1/Output
//   IMD_PLC/IMD_PLC Instance <-> Device 2 (EtherCAT)/MCC01_2_610A1 (EK1100)/610A2 (EK1122)/Box V (gantry B) (EP1008-0001)
//     PlcTask Inputs/MAIN.ProductHandling.GantryB.ixCollision <-> Channel 6/Input
//     PlcTask Inputs/MAIN.ProductHandling.GantryB.ixVacuumSensor[{1..5}] <-> Channel {1..5}/Input  (5 links)
//   IMD_PLC/IMD_PLC Instance <-> Device 2 (EtherCAT)/MCC01_2_610A1 (EK1100)/610A2 (EK1122)/Drive A-Belt / B-Spraybar (AX5201-0000-0203)
//     PlcTask Inputs/MAIN.InMoldDrying.ProductForming.SprayBarMotor.iDriveRef/aNetId <-> InfoData/AdsAddr/netId
//     PlcTask Inputs/MAIN.InMoldDrying.ProductForming.SprayBarMotor.iDriveRef/nDriveNo <-> InfoData/Chn1
//     PlcTask Inputs/MAIN.InMoldDrying.ProductForming.SprayBarMotor.iDriveRef/nSlaveAddr <-> InfoData/AdsAddr/port
//   IMD_PLC/IMD_PLC Instance <-> Device 2 (EtherCAT)/MCC01_2_610A1 (EK1100)/610A2 (EK1122)/Drive Gantry A (AX5203-0000-0203)
//     PlcTask Inputs/MAIN.ProductHandling.GantryA.HorizontalAxis.iDriveRef/aNetId <-> InfoData/AdsAddr/netId
//     PlcTask Inputs/MAIN.ProductHandling.GantryA.HorizontalAxis.iDriveRef/nDriveNo <-> InfoData/Chn0
//     PlcTask Inputs/MAIN.ProductHandling.GantryA.HorizontalAxis.iDriveRef/nSlaveAddr <-> InfoData/AdsAddr/port
//     PlcTask Inputs/MAIN.ProductHandling.GantryA.VerticalAxis.iDriveRef/aNetId <-> InfoData/AdsAddr/netId
//     PlcTask Inputs/MAIN.ProductHandling.GantryA.VerticalAxis.iDriveRef/nDriveNo <-> InfoData/Chn1
//     PlcTask Inputs/MAIN.ProductHandling.GantryA.VerticalAxis.iDriveRef/nSlaveAddr <-> InfoData/AdsAddr/port
//   IMD_PLC/IMD_PLC Instance <-> Device 2 (EtherCAT)/MCC01_2_610A1 (EK1100)/610A2 (EK1122)/Drive Gantry B (AX5203-0000-0203)
//     PlcTask Inputs/MAIN.ProductHandling.GantryB.HorizontalAxis.iDriveRef/aNetId <-> InfoData/AdsAddr/netId
//     PlcTask Inputs/MAIN.ProductHandling.GantryB.HorizontalAxis.iDriveRef/nDriveNo <-> InfoData/Chn0
//     PlcTask Inputs/MAIN.ProductHandling.GantryB.HorizontalAxis.iDriveRef/nSlaveAddr <-> InfoData/AdsAddr/port
//     PlcTask Inputs/MAIN.ProductHandling.GantryB.VerticalAxis.iDriveRef/aNetId <-> InfoData/AdsAddr/netId
//     PlcTask Inputs/MAIN.ProductHandling.GantryB.VerticalAxis.iDriveRef/nDriveNo <-> InfoData/Chn1
//     PlcTask Inputs/MAIN.ProductHandling.GantryB.VerticalAxis.iDriveRef/nSlaveAddr <-> InfoData/AdsAddr/port
//   IMD_PLC/IMD_PLC Instance <-> Device 2 (EtherCAT)/MCC01_2_610A1 (EK1100)/610A2 (EK1122)/EJBox (EP9128-0021)/JB_ (EP9128-1021)/Box AA (EP1008-0001)
//     PlcTask Inputs/MAIN.InMoldDrying.ProductForming.FeedingPulp.IxIsIn <-> Channel 3/Input
//     PlcTask Inputs/MAIN.InMoldDrying.ProductForming.FeedingPulp.IxIsOut <-> Channel 4/Input
//     PlcTask Inputs/MAIN.InMoldDrying.ProductForming.ixSprayBar_BackA <-> Channel 6/Input
//     PlcTask Inputs/MAIN.InMoldDrying.ProductForming.ixSprayBar_BackB <-> Channel 8/Input
//     PlcTask Inputs/MAIN.InMoldDrying.ProductForming.ixSprayBar_FrontA <-> Channel 5/Input
//     PlcTask Inputs/MAIN.InMoldDrying.ProductForming.ixSprayBar_FrontB <-> Channel 7/Input
//     PlcTask Inputs/MAIN.MainAirPressureSwitch <-> Channel 1/Input
//   IMD_PLC/IMD_PLC Instance <-> Device 2 (EtherCAT)/MCC01_2_610A1 (EK1100)/610A2 (EK1122)/EJBox (EP9128-0021)/JB_ (EP9128-1021)/Box B (EP2008-0001)
//     PlcTask Outputs/MAIN.InMoldDrying.HydraulicsMain.AccuDrainValve.Q <-> Channel 7/Output
//     PlcTask Outputs/MAIN.InMoldDrying.TopMoldA.BlowOff.Q <-> Channel 4/Output
//     PlcTask Outputs/MAIN.InMoldDrying.TopMoldA.Vacuum.Q <-> Channel 3/Output
//     PlcTask Outputs/MAIN.InMoldDrying.TopMoldB.BlowOff.Q <-> Channel 6/Output
//     PlcTask Outputs/MAIN.InMoldDrying.TopMoldB.Vacuum.Q <-> Channel 5/Output
//     PlcTask Outputs/MAIN.InMoldDrying.TransferMold.BlowOff.Q <-> Channel 1/Output
//     PlcTask Outputs/MAIN.InMoldDrying.TransferMold.Vacuum.Q <-> Channel 2/Output
//   IMD_PLC/IMD_PLC Instance <-> Device 2 (EtherCAT)/MCC01_2_610A1 (EK1100)/610A2 (EK1122)/EJBox (EP9128-0021)/JB_ (EP9128-1021)/Box C (EP2008-0001)
//     PlcTask Outputs/MAIN.InMoldDrying.BottomMoldA.Vacuum.Q <-> Channel 6/Output
//     PlcTask Outputs/MAIN.InMoldDrying.BottomMoldB.BlowOff.Q <-> Channel 7/Output
//     PlcTask Outputs/MAIN.InMoldDrying.ProductForming.FeedingPulp.QxIn <-> Channel 3/Output
//     PlcTask Outputs/MAIN.InMoldDrying.ProductForming.FlashSprayValve.Q <-> Channel 5/Output
//     PlcTask Outputs/MAIN.InMoldDrying.ProductForming.MoldBlowOff.Q <-> Channel 1/Output
//     PlcTask Outputs/MAIN.InMoldDrying.ProductForming.MoldVacuum.Q <-> Channel 2/Output
//     PlcTask Outputs/MAIN.InMoldDrying.ProductForming.WireSprayValve.Q <-> Channel 4/Output
//   IMD_PLC/IMD_PLC Instance <-> Device 2 (EtherCAT)/MCC01_2_610A1 (EK1100)/610A2 (EK1122)/EJBox (EP9128-0021)/JB_ (EP9128-1021)/Box D (EP2028-0001)
//     PlcTask Outputs/MAIN.InMoldDrying.ProductForming.PondHydraulicCilinder.HydraulicIn.Q <-> Channel 2/Output
//     PlcTask Outputs/MAIN.InMoldDrying.ProductForming.PondHydraulicCilinder.HydraulicOut.Q <-> Channel 1/Output
//     PlcTask Outputs/MAIN.InMoldDrying.ProductForming.PondHydraulicCilinder.HydraulicSlow.Q <-> Channel 3/Output
//   IMD_PLC/IMD_PLC Instance <-> Device 2 (EtherCAT)/MCC01_2_610A1 (EK1100)/610A2 (EK1122)/EJBox (EP9128-0021)/JB_ (EP9128-1021)/Box EF (EP2308-0001)
//     PlcTask Inputs/MAIN.InMoldDrying.BottomMoldA.HorizontalCilinder.IxIsIn <-> Channel 1/Input
//     PlcTask Inputs/MAIN.InMoldDrying.BottomMoldA.HorizontalCilinder.IxIsOut <-> Channel 2/Input
//     PlcTask Outputs/MAIN.InMoldDrying.BottomMoldA.HorizontalCilinder.QxIn <-> Channel 5/Output
//     PlcTask Outputs/MAIN.InMoldDrying.BottomMoldA.HorizontalCilinder.QxOut <-> Channel 6/Output
//   IMD_PLC/IMD_PLC Instance <-> Device 2 (EtherCAT)/MCC01_2_610A1 (EK1100)/610A2 (EK1122)/EJBox (EP9128-0021)/JB_ (EP9128-1021)/Box J (EP2008-0001)
//     PlcTask Outputs/MAIN.InMoldDrying.BottomMoldA.BlowOff.Q <-> Channel 2/Output
//     PlcTask Outputs/MAIN.InMoldDrying.BottomMoldB.Vacuum.Q <-> Channel 1/Output
//     PlcTask Outputs/MAIN.MainAirSupply.Q <-> Channel 4/Output
//   IMD_PLC/IMD_PLC Instance <-> Device 2 (EtherCAT)/MCC01_2_610A1 (EK1100)/610A2 (EK1122)/EJBox (EP9128-0021)/JB_ (EP9128-1021)/Box K (EP2008-0001)
//     PlcTask Outputs/MAIN.InMoldDrying.BottomMoldA.VacuumTakeout[{1..6}].Q <-> Channel {3..8}/Output  (6 links)
//     PlcTask Outputs/MAIN.InMoldDrying.BottomMoldA.VerticalCilinder.QxIn <-> Channel 1/Output
//     PlcTask Outputs/MAIN.InMoldDrying.BottomMoldA.VerticalCilinder.QxOut <-> Channel 2/Output
//   IMD_PLC/IMD_PLC Instance <-> Device 2 (EtherCAT)/MCC01_2_610A1 (EK1100)/610A2 (EK1122)/EJBox (EP9128-0021)/JB_ (EP9128-1021)/Box L (EP1008-0001)
//     PlcTask Inputs/MAIN.InMoldDrying.BottomMoldA.VacuumSensor[{1..6}] <-> Channel {3..8}/Input  (6 links)
//     PlcTask Inputs/MAIN.InMoldDrying.BottomMoldA.VerticalCilinder.IxIsIn <-> Channel 1/Input
//     PlcTask Inputs/MAIN.InMoldDrying.BottomMoldA.VerticalCilinder.IxIsOut <-> Channel 2/Input
//   IMD_PLC/IMD_PLC Instance <-> Device 2 (EtherCAT)/MCC01_2_610A1 (EK1100)/610A2 (EK1122)/EJBox (EP9128-0021)/JB_ (EP9128-1021)/Box Y1
//     PlcTask Inputs/MAIN.InMoldDrying.TopMoldA.HydraulicCilinder.BottomSidePressure.RawInput <-> AI Standard Channel 1/Value
//     PlcTask Inputs/MAIN.InMoldDrying.TopMoldA.HydraulicCilinder.RodSidePressure.RawInput <-> AI Standard Channel 2/Value
//     PlcTask Inputs/MAIN.InMoldDrying.TransferMold.HydraulicCilinder.BottomSidePressure.RawInput <-> AI Standard Channel 3/Value
//     PlcTask Inputs/MAIN.InMoldDrying.TransferMold.HydraulicCilinder.RodSidePressure.RawInput <-> AI Standard Channel 4/Value
//   IMD_PLC/IMD_PLC Instance <-> Device 2 (EtherCAT)/MCC01_2_610A1 (EK1100)/610A2 (EK1122)/EJBox (EP9128-0021)/JB_ (EP9128-1021)/Box Y2 (EP3174-0002)
//     PlcTask Inputs/MAIN.InMoldDrying.HydraulicsMain.MainSystemPressure.RawInput <-> AI Standard Channel 3/Value
//     PlcTask Inputs/MAIN.InMoldDrying.TopMoldB.HydraulicCilinder.BottomSidePressure.RawInput <-> AI Standard Channel 1/Value
//     PlcTask Inputs/MAIN.InMoldDrying.TopMoldB.HydraulicCilinder.RodSidePressure.RawInput <-> AI Standard Channel 2/Value
//   IMD_PLC/IMD_PLC Instance <-> Device 2 (EtherCAT)/MCC01_2_610A1 (EK1100)/610A2 (EK1122)/EJBox (EP9128-0021)/JB_BottomMoldB_GantryA (EP9128-2021)/Box HI (EP2308-0001)
//     PlcTask Inputs/MAIN.InMoldDrying.BottomMoldB.HorizontalCilinder.IxIsIn <-> Channel 1/Input
//     PlcTask Inputs/MAIN.InMoldDrying.BottomMoldB.HorizontalCilinder.IxIsOut <-> Channel 2/Input
//     PlcTask Outputs/MAIN.InMoldDrying.BottomMoldB.HorizontalCilinder.QxIn <-> Channel 6/Output
//     PlcTask Outputs/MAIN.InMoldDrying.BottomMoldB.HorizontalCilinder.QxOut <-> Channel 5/Output
//   IMD_PLC/IMD_PLC Instance <-> Device 2 (EtherCAT)/MCC01_2_610A1 (EK1100)/610A2 (EK1122)/EJBox (EP9128-0021)/JB_BottomMoldB_GantryA (EP9128-2021)/Box M (EP2008-0001)
//     PlcTask Outputs/MAIN.InMoldDrying.BottomMoldB.VacuumTakeout[{1..6}].Q <-> Channel {3..8}/Output  (6 links)
//     PlcTask Outputs/MAIN.InMoldDrying.BottomMoldB.VerticalCilinder.QxIn <-> Channel 1/Output
//     PlcTask Outputs/MAIN.InMoldDrying.BottomMoldB.VerticalCilinder.QxOut <-> Channel 2/Output
//   IMD_PLC/IMD_PLC Instance <-> Device 2 (EtherCAT)/MCC01_2_610A1 (EK1100)/610A2 (EK1122)/EJBox (EP9128-0021)/JB_BottomMoldB_GantryA (EP9128-2021)/Box N (EP1008-0001)
//     PlcTask Inputs/MAIN.InMoldDrying.BottomMoldB.VacuumSensor[{1..6}] <-> Channel {3..8}/Input  (6 links)
//     PlcTask Inputs/MAIN.InMoldDrying.BottomMoldB.VerticalCilinder.IxIsIn <-> Channel 1/Input
//     PlcTask Inputs/MAIN.InMoldDrying.BottomMoldB.VerticalCilinder.IxIsOut <-> Channel 2/Input
//   IMD_PLC/IMD_PLC Instance <-> Device 2 (EtherCAT)/MCC01_2_610A1 (EK1100)/610A2 (EK1122)/EJBox (EP9128-0021)/JB_BottomMoldB_GantryA (EP9128-2021)/Box O (EP1008-0001)
//     PlcTask Inputs/MAIN.ProductHandling.GantryA.ixEndLimitHorBack <-> Channel 2/Input
//     PlcTask Inputs/MAIN.ProductHandling.GantryA.ixEndLimitHorFront <-> Channel 1/Input
//   IMD_PLC/IMD_PLC Instance <-> Device 2 (EtherCAT)/MCC01_2_610A1 (EK1100)/610A2 (EK1122)/EJBox (EP9128-0021)/JB_BottomMoldB_GantryA (EP9128-2021)/Box P (EP1008-0001)
//     PlcTask Inputs/MAIN.ProductHandling.GantryA.ixEndLimitVertDown <-> Channel 2/Input
//     PlcTask Inputs/MAIN.ProductHandling.GantryA.ixEndLimitVertUp <-> Channel 1/Input
//   IMD_PLC/IMD_PLC Instance <-> Device 2 (EtherCAT)/MCC01_2_610A1 (EK1100)/610A2 (EK1122)/EJBox (EP9128-0021)/JB_BottomMoldB_GantryA (EP9128-2021)/Box Q1 (EP2008-0001)
//     PlcTask Outputs/MAIN.ProductHandling.GantryA.BlowOff[{1..4}].Q <-> Channel {2..8 step 2}/Output  (4 links)
//     PlcTask Outputs/MAIN.ProductHandling.GantryA.VacuumValve[{1..4}].Q <-> Channel {1..7 step 2}/Output  (4 links)
//   IMD_PLC/IMD_PLC Instance <-> Device 2 (EtherCAT)/MCC01_2_610A1 (EK1100)/610A2 (EK1122)/EJBox (EP9128-0021)/JB_BottomMoldB_GantryA (EP9128-2021)/Box Q2 (EP2008-0001)
//     PlcTask Outputs/MAIN.ProductHandling.GantryA.BlowOff[5].Q <-> Channel 2/Output
//     PlcTask Outputs/MAIN.ProductHandling.GantryA.VacuumValve[5].Q <-> Channel 1/Output
//   IMD_PLC/IMD_PLC Instance <-> Device 2 (EtherCAT)/MCC01_2_610A1 (EK1100)/610A2 (EK1122)/EJBox (EP9128-0021)/JB_BottomMoldB_GantryA (EP9128-2021)/Box R (EP1008-0001)
//     PlcTask Inputs/MAIN.ProductHandling.GantryA.ixCollision <-> Channel 6/Input
//     PlcTask Inputs/MAIN.ProductHandling.GantryA.ixVacuumSensor[{1..5}] <-> Channel {1..5}/Input  (5 links)
//   IMD_PLC/IMD_PLC Instance <-> Device 2 (EtherCAT)/MCC01_2_610A1 (EK1100)/610A2 (EK1122)/EJBox (EP9128-0021)/MachinePond (BTL7 EtherCAT)
//     PlcTask Inputs/MAIN.InMoldDrying.ProductForming.PondHydraulicCilinder.HydraulicPos.Magnet/CamState{1..4} <-> Module 1 (Position, speed, state, CAM and workarea)/Position, speed, state, CAM and workarea/CAM State {1..4}  (4 links)
//     PlcTask Inputs/MAIN.InMoldDrying.ProductForming.PondHydraulicCilinder.HydraulicPos.Magnet/PosAboveWorkAreaHighLimit <-> Module 1 (Position, speed, state, CAM and workarea)/Position, speed, state, CAM and workarea/Position above work area high limit
//     PlcTask Inputs/MAIN.InMoldDrying.ProductForming.PondHydraulicCilinder.HydraulicPos.Magnet/PosBelowWorkAreaLowLimit <-> Module 1 (Position, speed, state, CAM and workarea)/Position, speed, state, CAM and workarea/Position below work area low limit
//     PlcTask Inputs/MAIN.InMoldDrying.ProductForming.PondHydraulicCilinder.HydraulicPos.Magnet/PosMarkerFailure <-> Module 1 (Position, speed, state, CAM and workarea)/Position, speed, state, CAM and workarea/Position marker failure
//     PlcTask Inputs/MAIN.InMoldDrying.ProductForming.PondHydraulicCilinder.HydraulicPos.Magnet/Position <-> Module 1 (Position, speed, state, CAM and workarea)/Position, speed, state, CAM and workarea/Position
//     PlcTask Inputs/MAIN.InMoldDrying.ProductForming.PondHydraulicCilinder.HydraulicPos.Magnet/Speed <-> Module 1 (Position, speed, state, CAM and workarea)/Position, speed, state, CAM and workarea/Speed
//   IMD_PLC/IMD_PLC Instance <-> Device 2 (EtherCAT)/MCC01_2_610A1 (EK1100)/610A2 (EK1122)/EJBox (EP9128-0021)/RIO_600A1 (EK1100)/RIO_600A11 (EL1904)
//     PlcTask Inputs/MAIN.ixEmStopImdBack[0] <-> Module 1 (FSOES)/TxPDO/FSOE/InputChannel3
//     PlcTask Inputs/MAIN.ixEmStopImdBack[1] <-> Module 1 (FSOES)/TxPDO/FSOE/InputChannel4
//     PlcTask Inputs/MAIN.ixEmStopImdFront[0] <-> Module 1 (FSOES)/TxPDO/FSOE/InputChannel1
//     PlcTask Inputs/MAIN.ixEmStopImdFront[1] <-> Module 1 (FSOES)/TxPDO/FSOE/InputChannel2
//   IMD_PLC/IMD_PLC Instance <-> Device 2 (EtherCAT)/MCC01_2_610A1 (EK1100)/610A2 (EK1122)/EJBox (EP9128-0021)/RIO_600A1 (EK1100)/RIO_600A12 (EL1904)
//     PlcTask Inputs/MAIN.ixEmStopGantryA_Back[0] <-> Module 1 (FSOES)/TxPDO/FSOE/InputChannel3
//     PlcTask Inputs/MAIN.ixEmStopGantryA_Back[1] <-> Module 1 (FSOES)/TxPDO/FSOE/InputChannel4
//     PlcTask Inputs/MAIN.ixEmStopGantryA_Front[0] <-> Module 1 (FSOES)/TxPDO/FSOE/InputChannel1
//     PlcTask Inputs/MAIN.ixEmStopGantryA_Front[1] <-> Module 1 (FSOES)/TxPDO/FSOE/InputChannel2
//   IMD_PLC/IMD_PLC Instance <-> Device 2 (EtherCAT)/MCC01_2_610A1 (EK1100)/610A2 (EK1122)/EJBox (EP9128-0021)/RIO_600A1 (EK1100)/RIO_600A13 (EL1904)
//     PlcTask Inputs/MAIN.ixEmStopGantryB_Back[0] <-> Module 1 (FSOES)/TxPDO/FSOE/InputChannel3
//     PlcTask Inputs/MAIN.ixEmStopGantryB_Back[1] <-> Module 1 (FSOES)/TxPDO/FSOE/InputChannel4
//     PlcTask Inputs/MAIN.ixEmStopGantryB_Front[0] <-> Module 1 (FSOES)/TxPDO/FSOE/InputChannel1
//     PlcTask Inputs/MAIN.ixEmStopGantryB_Front[1] <-> Module 1 (FSOES)/TxPDO/FSOE/InputChannel2
//   IMD_PLC/IMD_PLC Instance <-> Device 2 (EtherCAT)/MCC01_2_610A1 (EK1100)/610A2 (EK1122)/EJBox (EP9128-0021)/RIO_600A1 (EK1100)/RIO_600A16 (EL1904)
//     PlcTask Inputs/MAIN.ixSafetyFrontDoorLeft[0] <-> Module 1 (FSOES)/TxPDO/FSOE/InputChannel1
//     PlcTask Inputs/MAIN.ixSafetyFrontDoorLeft[1] <-> Module 1 (FSOES)/TxPDO/FSOE/InputChannel2
//     PlcTask Inputs/MAIN.ixSafetyFrontDoorMiddle[0] <-> Module 1 (FSOES)/TxPDO/FSOE/InputChannel3
//     PlcTask Inputs/MAIN.ixSafetyFrontDoorMiddle[1] <-> Module 1 (FSOES)/TxPDO/FSOE/InputChannel4
//   IMD_PLC/IMD_PLC Instance <-> Device 2 (EtherCAT)/MCC01_2_610A1 (EK1100)/610A2 (EK1122)/EJBox (EP9128-0021)/RIO_600A1 (EK1100)/RIO_600A17 (EL1904)
//     PlcTask Inputs/MAIN.ixSafetyFrontDoorRight[0] <-> Module 1 (FSOES)/TxPDO/FSOE/InputChannel1
//     PlcTask Inputs/MAIN.ixSafetyFrontDoorRight[1] <-> Module 1 (FSOES)/TxPDO/FSOE/InputChannel2
//   IMD_PLC/IMD_PLC Instance <-> Device 2 (EtherCAT)/MCC01_2_610A1 (EK1100)/610A2 (EK1122)/EJBox (EP9128-0021)/RIO_600A1 (EK1100)/RIO_600A2 (EL1804)
//     PlcTask Inputs/MAIN.ixDoorReqImdBack <-> Channel 4/Input
//     PlcTask Inputs/MAIN.ixDoorReqImdFront <-> Channel 2/Input
//     PlcTask Inputs/MAIN.ixResetImdBack <-> Channel 3/Input
//     PlcTask Inputs/MAIN.ixResetImdFront <-> Channel 1/Input
//   IMD_PLC/IMD_PLC Instance <-> Device 2 (EtherCAT)/MCC01_2_610A1 (EK1100)/610A2 (EK1122)/EJBox (EP9128-0021)/RIO_600A1 (EK1100)/RIO_600A20 (EL1904)
//     PlcTask Inputs/MAIN.ixSafetyBackDoorLeft1[0] <-> Module 1 (FSOES)/TxPDO/FSOE/InputChannel1
//     PlcTask Inputs/MAIN.ixSafetyBackDoorLeft1[1] <-> Module 1 (FSOES)/TxPDO/FSOE/InputChannel2
//     PlcTask Inputs/MAIN.ixSafetyBackDoorLeft2[0] <-> Module 1 (FSOES)/TxPDO/FSOE/InputChannel3
//     PlcTask Inputs/MAIN.ixSafetyBackDoorLeft2[1] <-> Module 1 (FSOES)/TxPDO/FSOE/InputChannel4
//   IMD_PLC/IMD_PLC Instance <-> Device 2 (EtherCAT)/MCC01_2_610A1 (EK1100)/610A2 (EK1122)/EJBox (EP9128-0021)/RIO_600A1 (EK1100)/RIO_600A21 (EL1904)
//     PlcTask Inputs/MAIN.ixSafetyBackDoorMiddle3[0] <-> Module 1 (FSOES)/TxPDO/FSOE/InputChannel1
//     PlcTask Inputs/MAIN.ixSafetyBackDoorMiddle3[1] <-> Module 1 (FSOES)/TxPDO/FSOE/InputChannel2
//     PlcTask Inputs/MAIN.ixSafetyBackDoorMiddle4[0] <-> Module 1 (FSOES)/TxPDO/FSOE/InputChannel3
//     PlcTask Inputs/MAIN.ixSafetyBackDoorMiddle4[1] <-> Module 1 (FSOES)/TxPDO/FSOE/InputChannel4
//   IMD_PLC/IMD_PLC Instance <-> Device 2 (EtherCAT)/MCC01_2_610A1 (EK1100)/610A2 (EK1122)/EJBox (EP9128-0021)/RIO_600A1 (EK1100)/RIO_600A22 (EL1904)
//     PlcTask Inputs/MAIN.ixSafetyBackDoorRight5[0] <-> Module 1 (FSOES)/TxPDO/FSOE/InputChannel1
//     PlcTask Inputs/MAIN.ixSafetyBackDoorRight5[1] <-> Module 1 (FSOES)/TxPDO/FSOE/InputChannel2
//     PlcTask Inputs/MAIN.ixSafetyBackDoorRight6[0] <-> Module 1 (FSOES)/TxPDO/FSOE/InputChannel3
//     PlcTask Inputs/MAIN.ixSafetyBackDoorRight6[1] <-> Module 1 (FSOES)/TxPDO/FSOE/InputChannel4
//   IMD_PLC/IMD_PLC Instance <-> Device 2 (EtherCAT)/MCC01_2_610A1 (EK1100)/610A2 (EK1122)/EJBox (EP9128-0021)/RIO_600A1 (EK1100)/RIO_600A23 (EL1904)
//     PlcTask Inputs/MAIN.ixSafetyGantryA_FrontDoorLeft[0] <-> Module 1 (FSOES)/TxPDO/FSOE/InputChannel1
//     PlcTask Inputs/MAIN.ixSafetyGantryA_FrontDoorLeft[1] <-> Module 1 (FSOES)/TxPDO/FSOE/InputChannel2
//     PlcTask Inputs/MAIN.ixSafetyGantryA_FrontDoorRight[0] <-> Module 1 (FSOES)/TxPDO/FSOE/InputChannel3
//     PlcTask Inputs/MAIN.ixSafetyGantryA_FrontDoorRight[1] <-> Module 1 (FSOES)/TxPDO/FSOE/InputChannel4
//   IMD_PLC/IMD_PLC Instance <-> Device 2 (EtherCAT)/MCC01_2_610A1 (EK1100)/610A2 (EK1122)/EJBox (EP9128-0021)/RIO_600A1 (EK1100)/RIO_600A24 (EL1904)
//     PlcTask Inputs/MAIN.ixSafetyGantryA_BackDoor[0] <-> Module 1 (FSOES)/TxPDO/FSOE/InputChannel1
//     PlcTask Inputs/MAIN.ixSafetyGantryA_BackDoor[1] <-> Module 1 (FSOES)/TxPDO/FSOE/InputChannel2
//   IMD_PLC/IMD_PLC Instance <-> Device 2 (EtherCAT)/MCC01_2_610A1 (EK1100)/610A2 (EK1122)/EJBox (EP9128-0021)/RIO_600A1 (EK1100)/RIO_600A25 (EL1904)
//     PlcTask Inputs/MAIN.ixSafetyGantryB_FrontDoorLeft[0] <-> Module 1 (FSOES)/TxPDO/FSOE/InputChannel1
//     PlcTask Inputs/MAIN.ixSafetyGantryB_FrontDoorLeft[1] <-> Module 1 (FSOES)/TxPDO/FSOE/InputChannel2
//     PlcTask Inputs/MAIN.ixSafetyGantryB_FrontDoorRight[0] <-> Module 1 (FSOES)/TxPDO/FSOE/InputChannel3
//     PlcTask Inputs/MAIN.ixSafetyGantryB_FrontDoorRight[1] <-> Module 1 (FSOES)/TxPDO/FSOE/InputChannel4
//   IMD_PLC/IMD_PLC Instance <-> Device 2 (EtherCAT)/MCC01_2_610A1 (EK1100)/610A2 (EK1122)/EJBox (EP9128-0021)/RIO_600A1 (EK1100)/RIO_600A26 (EL1904)
//     PlcTask Inputs/MAIN.ixSafetyGantryB_BackDoor[0] <-> Module 1 (FSOES)/TxPDO/FSOE/InputChannel1
//     PlcTask Inputs/MAIN.ixSafetyGantryB_BackDoor[1] <-> Module 1 (FSOES)/TxPDO/FSOE/InputChannel2
//   IMD_PLC/IMD_PLC Instance <-> Device 2 (EtherCAT)/MCC01_2_610A1 (EK1100)/610A2 (EK1122)/EJBox (EP9128-0021)/RIO_600A1 (EK1100)/RIO_600A3 (EL1804)
//     PlcTask Inputs/MAIN.ixDoorReqGantryA_Back <-> Channel 4/Input
//     PlcTask Inputs/MAIN.ixDoorReqGantryA_Front <-> Channel 2/Input
//     PlcTask Inputs/MAIN.ixResetGantryA_Back <-> Channel 3/Input
//     PlcTask Inputs/MAIN.ixResetGantryA_Front <-> Channel 1/Input
//   IMD_PLC/IMD_PLC Instance <-> Device 2 (EtherCAT)/MCC01_2_610A1 (EK1100)/610A2 (EK1122)/EJBox (EP9128-0021)/RIO_600A1 (EK1100)/RIO_600A4 (EL1804)
//     PlcTask Inputs/MAIN.ixDoorReqGantryB_Back <-> Channel 4/Input
//     PlcTask Inputs/MAIN.ixDoorReqGantryB_Front <-> Channel 2/Input
//     PlcTask Inputs/MAIN.ixResetGantryB_Back <-> Channel 3/Input
//     PlcTask Inputs/MAIN.ixResetGantryB_Front <-> Channel 1/Input
//   IMD_PLC/IMD_PLC Instance <-> Device 2 (EtherCAT)/MCC01_2_610A1 (EK1100)/610A2 (EK1122)/EJBox (EP9128-0021)/RIO_600A1 (EK1100)/RIO_600A7 (EL2808)
//     PlcTask Outputs/MAIN.qxLightDoorReqGantryA_Back <-> Channel 8/Output
//     PlcTask Outputs/MAIN.qxLightDoorReqGantryA_Front <-> Channel 6/Output
//     PlcTask Outputs/MAIN.qxLightDoorReqImdBack <-> Channel 4/Output
//     PlcTask Outputs/MAIN.qxLightDoorReqImdFront <-> Channel 2/Output
//     PlcTask Outputs/MAIN.qxLightEmStopGantryA_Back <-> Channel 7/Output
//     PlcTask Outputs/MAIN.qxLightEmStopGantryA_Front <-> Channel 5/Output
//     PlcTask Outputs/MAIN.qxLightEmStopImdBack <-> Channel 3/Output
//     PlcTask Outputs/MAIN.qxLightEmStopImdFront <-> Channel 1/Output
//   IMD_PLC/IMD_PLC Instance <-> Device 2 (EtherCAT)/MCC01_2_610A1 (EK1100)/610A2 (EK1122)/EJBox (EP9128-0021)/RIO_600A1 (EK1100)/RIO_600A8 (EL2808)
//     PlcTask Outputs/MAIN.qxLightDoorReqGantryB_Back <-> Channel 4/Output
//     PlcTask Outputs/MAIN.qxLightDoorReqGantryB_Front <-> Channel 2/Output
//     PlcTask Outputs/MAIN.qxLightEmStopGantryB_Back <-> Channel 3/Output
//     PlcTask Outputs/MAIN.qxLightEmStopGantryB_Front <-> Channel 1/Output
//   IMD_PLC/IMD_PLC Instance <-> Device 2 (EtherCAT)/MCC01_2_610A1 (EK1100)/610A2 (EK1122)/EJBox (EP9128-0021)/RIO_600A1 (EK1100)/RIO_600A9 (EL2808)
//     PlcTask Outputs/MAIN.qxAlarmHorn <-> Channel 4/Output
//     PlcTask Outputs/MAIN.qxLightGreen <-> Channel 1/Output
//     PlcTask Outputs/MAIN.qxLightRed <-> Channel 3/Output
//     PlcTask Outputs/MAIN.qxLightYellow <-> Channel 2/Output
//   IMD_PLC/IMD_PLC Instance <-> Device 2 (EtherCAT)/MCC01_2_610A1 (EK1100)/610A2 (EK1122)/EJBox (EP9128-0021)/TopMoldA (BTL7 EtherCAT)
//     PlcTask Inputs/MAIN.InMoldDrying.TopMoldA.HydraulicCilinder.HydraulicPos.Magnet/CamState{1..4} <-> Module 1 (Position, speed, state, CAM and workarea)/Position, speed, state, CAM and workarea/CAM State {1..4}  (4 links)
//     PlcTask Inputs/MAIN.InMoldDrying.TopMoldA.HydraulicCilinder.HydraulicPos.Magnet/PosAboveWorkAreaHighLimit <-> Module 1 (Position, speed, state, CAM and workarea)/Position, speed, state, CAM and workarea/Position above work area high limit
//     PlcTask Inputs/MAIN.InMoldDrying.TopMoldA.HydraulicCilinder.HydraulicPos.Magnet/PosBelowWorkAreaLowLimit <-> Module 1 (Position, speed, state, CAM and workarea)/Position, speed, state, CAM and workarea/Position below work area low limit
//     PlcTask Inputs/MAIN.InMoldDrying.TopMoldA.HydraulicCilinder.HydraulicPos.Magnet/PosMarkerFailure <-> Module 1 (Position, speed, state, CAM and workarea)/Position, speed, state, CAM and workarea/Position marker failure
//     PlcTask Inputs/MAIN.InMoldDrying.TopMoldA.HydraulicCilinder.HydraulicPos.Magnet/Position <-> Module 1 (Position, speed, state, CAM and workarea)/Position, speed, state, CAM and workarea/Position
//     PlcTask Inputs/MAIN.InMoldDrying.TopMoldA.HydraulicCilinder.HydraulicPos.Magnet/Speed <-> Module 1 (Position, speed, state, CAM and workarea)/Position, speed, state, CAM and workarea/Speed
//   IMD_PLC/IMD_PLC Instance <-> Device 2 (EtherCAT)/MCC01_2_610A1 (EK1100)/610A2 (EK1122)/EJBox (EP9128-0021)/TopMoldB (BTL7 EtherCAT)
//     PlcTask Inputs/MAIN.InMoldDrying.TopMoldB.HydraulicCilinder.HydraulicPos.Magnet/CamState{1..4} <-> Module 1 (Position, speed, state, CAM and workarea)/Position, speed, state, CAM and workarea/CAM State {1..4}  (4 links)
//     PlcTask Inputs/MAIN.InMoldDrying.TopMoldB.HydraulicCilinder.HydraulicPos.Magnet/PosAboveWorkAreaHighLimit <-> Module 1 (Position, speed, state, CAM and workarea)/Position, speed, state, CAM and workarea/Position above work area high limit
//     PlcTask Inputs/MAIN.InMoldDrying.TopMoldB.HydraulicCilinder.HydraulicPos.Magnet/PosBelowWorkAreaLowLimit <-> Module 1 (Position, speed, state, CAM and workarea)/Position, speed, state, CAM and workarea/Position below work area low limit
//     PlcTask Inputs/MAIN.InMoldDrying.TopMoldB.HydraulicCilinder.HydraulicPos.Magnet/PosMarkerFailure <-> Module 1 (Position, speed, state, CAM and workarea)/Position, speed, state, CAM and workarea/Position marker failure
//     PlcTask Inputs/MAIN.InMoldDrying.TopMoldB.HydraulicCilinder.HydraulicPos.Magnet/Position <-> Module 1 (Position, speed, state, CAM and workarea)/Position, speed, state, CAM and workarea/Position
//     PlcTask Inputs/MAIN.InMoldDrying.TopMoldB.HydraulicCilinder.HydraulicPos.Magnet/Speed <-> Module 1 (Position, speed, state, CAM and workarea)/Position, speed, state, CAM and workarea/Speed
//   IMD_PLC/IMD_PLC Instance <-> Device 2 (EtherCAT)/MCC01_2_610A1 (EK1100)/610A2 (EK1122)/EJBox (EP9128-0021)/TransferMold (BTL7 EtherCAT)
//     PlcTask Inputs/MAIN.InMoldDrying.TransferMold.HydraulicCilinder.HydraulicPos.Magnet/CamState{1..4} <-> Module 1 (Position, speed, state, CAM and workarea)/Position, speed, state, CAM and workarea/CAM State {1..4}  (4 links)
//     PlcTask Inputs/MAIN.InMoldDrying.TransferMold.HydraulicCilinder.HydraulicPos.Magnet/PosAboveWorkAreaHighLimit <-> Module 1 (Position, speed, state, CAM and workarea)/Position, speed, state, CAM and workarea/Position above work area high limit
//     PlcTask Inputs/MAIN.InMoldDrying.TransferMold.HydraulicCilinder.HydraulicPos.Magnet/PosBelowWorkAreaLowLimit <-> Module 1 (Position, speed, state, CAM and workarea)/Position, speed, state, CAM and workarea/Position below work area low limit
//     PlcTask Inputs/MAIN.InMoldDrying.TransferMold.HydraulicCilinder.HydraulicPos.Magnet/PosMarkerFailure <-> Module 1 (Position, speed, state, CAM and workarea)/Position, speed, state, CAM and workarea/Position marker failure
//     PlcTask Inputs/MAIN.InMoldDrying.TransferMold.HydraulicCilinder.HydraulicPos.Magnet/Position <-> Module 1 (Position, speed, state, CAM and workarea)/Position, speed, state, CAM and workarea/Position
//     PlcTask Inputs/MAIN.InMoldDrying.TransferMold.HydraulicCilinder.HydraulicPos.Magnet/Speed <-> Module 1 (Position, speed, state, CAM and workarea)/Position, speed, state, CAM and workarea/Speed
//   IMD_PLC/IMD_PLC Instance <-> Device 2 (EtherCAT)/MCC01_2_610A1 (EK1100)/610A4 (EL3403)
//     PlcTask Inputs/MAIN.L1/iwActivePower <-> PM Inputs Channel 1/Active power
//     PlcTask Inputs/MAIN.L2/iwActivePower <-> PM Inputs Channel 2/Active power
//     PlcTask Inputs/MAIN.L3/iwActivePower <-> PM Inputs Channel 3/Active power
//     PlcTask Inputs/MAIN.L1/iwCurrent <-> PM Inputs Channel 1/Current
//     PlcTask Inputs/MAIN.L2/iwCurrent <-> PM Inputs Channel 2/Current
//     PlcTask Inputs/MAIN.L3/iwCurrent <-> PM Inputs Channel 3/Current
//     PlcTask Inputs/MAIN.L1/iwIndex <-> PM Inputs Channel 1/Index
//     PlcTask Inputs/MAIN.L2/iwIndex <-> PM Inputs Channel 2/Index
//     PlcTask Inputs/MAIN.L3/iwIndex <-> PM Inputs Channel 3/Index
//     PlcTask Inputs/MAIN.L1/iwVariantValue <-> PM Inputs Channel 1/Variant value
//     PlcTask Inputs/MAIN.L2/iwVariantValue <-> PM Inputs Channel 2/Variant value
//     PlcTask Inputs/MAIN.L3/iwVariantValue <-> PM Inputs Channel 3/Variant value
//     PlcTask Inputs/MAIN.L1/iwVoltage <-> PM Inputs Channel 1/Voltage
//     PlcTask Inputs/MAIN.L2/iwVoltage <-> PM Inputs Channel 2/Voltage
//     PlcTask Inputs/MAIN.L3/iwVoltage <-> PM Inputs Channel 3/Voltage
//     PlcTask Inputs/MAIN.L1/ixPDOToggle <-> PM Inputs Channel 1/TxPDO Toggle
//     PlcTask Inputs/MAIN.L2/ixPDOToggle <-> PM Inputs Channel 2/TxPDO Toggle
//     PlcTask Inputs/MAIN.L3/ixPDOToggle <-> PM Inputs Channel 3/TxPDO Toggle
//   IMD_PLC/IMD_PLC Instance <-> Device 2 (EtherCAT)/MCC01_2_610A1 (EK1100)/610A5 (EL3202)
//     PlcTask Inputs/MAIN.InMoldDrying.TopMoldA.HeatingZone[1].FB_Temperature.RawInput <-> RTD Inputs Channel 1/Value
//     PlcTask Inputs/MAIN.InMoldDrying.TopMoldA.HeatingZone[2].FB_Temperature.RawInput <-> RTD Inputs Channel 2/Value
//     PlcTask Inputs/MAIN.InMoldDrying.TopMoldA.HeatingZone[1].FB_Temperature.Status <-> RTD Inputs Channel 1/Status
//     PlcTask Inputs/MAIN.InMoldDrying.TopMoldA.HeatingZone[2].FB_Temperature.Status <-> RTD Inputs Channel 2/Status
//   IMD_PLC/IMD_PLC Instance <-> Device 2 (EtherCAT)/MCC01_2_610A1 (EK1100)/610A6 (EL3202)
//     PlcTask Inputs/MAIN.InMoldDrying.TopMoldA.HeatingZone[3].FB_Temperature.RawInput <-> RTD Inputs Channel 1/Value
//     PlcTask Inputs/MAIN.InMoldDrying.TopMoldA.HeatingZone[4].FB_Temperature.RawInput <-> RTD Inputs Channel 2/Value
//     PlcTask Inputs/MAIN.InMoldDrying.TopMoldA.HeatingZone[3].FB_Temperature.Status <-> RTD Inputs Channel 1/Status
//     PlcTask Inputs/MAIN.InMoldDrying.TopMoldA.HeatingZone[4].FB_Temperature.Status <-> RTD Inputs Channel 2/Status
//   IMD_PLC/IMD_PLC Instance <-> Device 2 (EtherCAT)/MCC01_2_610A1 (EK1100)/610A7 (EL3202)
//     PlcTask Inputs/MAIN.InMoldDrying.TopMoldA.HeatingZone[5].FB_Temperature.RawInput <-> RTD Inputs Channel 1/Value
//     PlcTask Inputs/MAIN.InMoldDrying.TopMoldA.HeatingZone[6].FB_Temperature.RawInput <-> RTD Inputs Channel 2/Value
//     PlcTask Inputs/MAIN.InMoldDrying.TopMoldA.HeatingZone[5].FB_Temperature.Status <-> RTD Inputs Channel 1/Status
//     PlcTask Inputs/MAIN.InMoldDrying.TopMoldA.HeatingZone[6].FB_Temperature.Status <-> RTD Inputs Channel 2/Status
//   IMD_PLC/IMD_PLC Instance <-> Device 2 (EtherCAT)/MCC01_2_610A1 (EK1100)/610A8 (EL3202)
//     PlcTask Inputs/MAIN.InMoldDrying.BottomMoldA.HeatingZone[1].FB_Temperature.RawInput <-> RTD Inputs Channel 1/Value
//     PlcTask Inputs/MAIN.InMoldDrying.BottomMoldA.HeatingZone[2].FB_Temperature.RawInput <-> RTD Inputs Channel 2/Value
//     PlcTask Inputs/MAIN.InMoldDrying.BottomMoldA.HeatingZone[1].FB_Temperature.Status <-> RTD Inputs Channel 1/Status
//     PlcTask Inputs/MAIN.InMoldDrying.BottomMoldA.HeatingZone[2].FB_Temperature.Status <-> RTD Inputs Channel 2/Status
//   IMD_PLC/IMD_PLC Instance <-> Device 2 (EtherCAT)/MCC01_2_610A1 (EK1100)/610A9 (EL3202)
//     PlcTask Inputs/MAIN.InMoldDrying.BottomMoldA.HeatingZone[3].FB_Temperature.RawInput <-> RTD Inputs Channel 1/Value
//     PlcTask Inputs/MAIN.InMoldDrying.BottomMoldA.HeatingZone[4].FB_Temperature.RawInput <-> RTD Inputs Channel 2/Value
//     PlcTask Inputs/MAIN.InMoldDrying.BottomMoldA.HeatingZone[3].FB_Temperature.Status <-> RTD Inputs Channel 1/Status
//     PlcTask Inputs/MAIN.InMoldDrying.BottomMoldA.HeatingZone[4].FB_Temperature.Status <-> RTD Inputs Channel 2/Status
//   IMD_PLC/IMD_PLC Instance <-> Device 2 (EtherCAT)/MCC01_600A1 (EK1100)/600A16 (EL1809)
//     PlcTask Inputs/MAIN.ix24VoltError1 <-> Channel 15/Input
//     PlcTask Inputs/MAIN.ix24VoltError2 <-> Channel 16/Input
//   IMD_PLC/IMD_PLC Instance <-> Device 2 (EtherCAT)/MCC01_600A1 (EK1100)/600A19 (EL1809)
//     PlcTask Inputs/MAIN.InMoldDrying.BottomMoldA.HeatingZone[{1..6}].ixThermal <-> Channel {7..12}/Input  (6 links)
//     PlcTask Inputs/MAIN.InMoldDrying.TopMoldA.HeatingZone[{1..6}].ixThermal <-> Channel {1..6}/Input  (6 links)
//   IMD_PLC/IMD_PLC Instance <-> Device 2 (EtherCAT)/MCC01_600A1 (EK1100)/600A20 (EL1809)
//     PlcTask Inputs/MAIN.InMoldDrying.BottomMoldB.HeatingZone[{1..6}].ixThermal <-> Channel {7..12}/Input  (6 links)
//     PlcTask Inputs/MAIN.InMoldDrying.TopMoldB.HeatingZone[{1..6}].ixThermal <-> Channel {1..6}/Input  (6 links)
//   IMD_PLC/IMD_PLC Instance <-> Device 2 (EtherCAT)/MCC01_600A1 (EK1100)/600A21 (EL1809)
//     PlcTask Inputs/MAIN.InMoldDrying.ProductForming.ixCssHasAnError <-> Channel 12/Input
//     PlcTask Inputs/MAIN.InMoldDrying.ProductForming.ixPulpTank01 <-> Channel 9/Input
//     PlcTask Inputs/MAIN.InMoldDrying.ProductForming.ixPulpTank02 <-> Channel 10/Input
//   IMD_PLC/IMD_PLC Instance <-> Device 2 (EtherCAT)/MCC01_600A1 (EK1100)/600A23 (EL2809)
//     PlcTask Outputs/MAIN.InMoldDrying.TopMoldA.HeatingZone[1].qxPWMOut1 <-> Channel 1/Output
//     PlcTask Outputs/MAIN.InMoldDrying.TopMoldA.HeatingZone[1].qxPWMOut2 <-> Channel 2/Output
//     PlcTask Outputs/MAIN.InMoldDrying.TopMoldA.HeatingZone[1].qxPWMOut3 <-> Channel 3/Output
//     PlcTask Outputs/MAIN.InMoldDrying.TopMoldA.HeatingZone[2].qxPWMOut1 <-> Channel 4/Output
//     PlcTask Outputs/MAIN.InMoldDrying.TopMoldA.HeatingZone[2].qxPWMOut2 <-> Channel 5/Output
//     PlcTask Outputs/MAIN.InMoldDrying.TopMoldA.HeatingZone[2].qxPWMOut3 <-> Channel 6/Output
//     PlcTask Outputs/MAIN.InMoldDrying.TopMoldA.HeatingZone[3].qxPWMOut1 <-> Channel 7/Output
//     PlcTask Outputs/MAIN.InMoldDrying.TopMoldA.HeatingZone[3].qxPWMOut2 <-> Channel 8/Output
//     PlcTask Outputs/MAIN.InMoldDrying.TopMoldA.HeatingZone[3].qxPWMOut3 <-> Channel 9/Output
//     PlcTask Outputs/MAIN.InMoldDrying.TopMoldA.HeatingZone[4].qxPWMOut1 <-> Channel 10/Output
//     PlcTask Outputs/MAIN.InMoldDrying.TopMoldA.HeatingZone[4].qxPWMOut2 <-> Channel 11/Output
//     PlcTask Outputs/MAIN.InMoldDrying.TopMoldA.HeatingZone[4].qxPWMOut3 <-> Channel 12/Output
//     PlcTask Outputs/MAIN.InMoldDrying.TopMoldA.HeatingZone[5].qxPWMOut1 <-> Channel 13/Output
//     PlcTask Outputs/MAIN.InMoldDrying.TopMoldA.HeatingZone[5].qxPWMOut2 <-> Channel 14/Output
//     PlcTask Outputs/MAIN.InMoldDrying.TopMoldA.HeatingZone[5].qxPWMOut3 <-> Channel 15/Output
//   IMD_PLC/IMD_PLC Instance <-> Device 2 (EtherCAT)/MCC01_600A1 (EK1100)/600A24 (EL2809)
//     PlcTask Outputs/MAIN.InMoldDrying.BottomMoldA.HeatingZone[1].qxPWMOut1 <-> Channel 5/Output
//     PlcTask Outputs/MAIN.InMoldDrying.BottomMoldA.HeatingZone[1].qxPWMOut2 <-> Channel 6/Output
//     PlcTask Outputs/MAIN.InMoldDrying.BottomMoldA.HeatingZone[1].qxPWMOut3 <-> Channel 7/Output
//     PlcTask Outputs/MAIN.InMoldDrying.BottomMoldA.HeatingZone[2].qxPWMOut1 <-> Channel 8/Output
//     PlcTask Outputs/MAIN.InMoldDrying.BottomMoldA.HeatingZone[2].qxPWMOut2 <-> Channel 9/Output
//     PlcTask Outputs/MAIN.InMoldDrying.BottomMoldA.HeatingZone[2].qxPWMOut3 <-> Channel 10/Output
//     PlcTask Outputs/MAIN.InMoldDrying.BottomMoldA.HeatingZone[3].qxPWMOut1 <-> Channel 11/Output
//     PlcTask Outputs/MAIN.InMoldDrying.BottomMoldA.HeatingZone[3].qxPWMOut2 <-> Channel 12/Output
//     PlcTask Outputs/MAIN.InMoldDrying.BottomMoldA.HeatingZone[3].qxPWMOut3 <-> Channel 13/Output
//     PlcTask Outputs/MAIN.InMoldDrying.BottomMoldA.HeatingZone[4].qxPWMOut1 <-> Channel 14/Output
//     PlcTask Outputs/MAIN.InMoldDrying.BottomMoldA.HeatingZone[4].qxPWMOut2 <-> Channel 15/Output
//     PlcTask Outputs/MAIN.InMoldDrying.BottomMoldA.HeatingZone[4].qxPWMOut3 <-> Channel 16/Output
//     PlcTask Outputs/MAIN.InMoldDrying.TopMoldA.HeatingZone[6].qxPWMOut1 <-> Channel 1/Output
//     PlcTask Outputs/MAIN.InMoldDrying.TopMoldA.HeatingZone[6].qxPWMOut2 <-> Channel 2/Output
//     PlcTask Outputs/MAIN.InMoldDrying.TopMoldA.HeatingZone[6].qxPWMOut3 <-> Channel 3/Output
//   IMD_PLC/IMD_PLC Instance <-> Device 2 (EtherCAT)/MCC01_600A1 (EK1100)/600A25 (EL2809)
//     PlcTask Outputs/MAIN.InMoldDrying.BottomMoldA.HeatingZone[5].qxPWMOut1 <-> Channel 1/Output
//     PlcTask Outputs/MAIN.InMoldDrying.BottomMoldA.HeatingZone[5].qxPWMOut2 <-> Channel 2/Output
//     PlcTask Outputs/MAIN.InMoldDrying.BottomMoldA.HeatingZone[5].qxPWMOut3 <-> Channel 3/Output
//     PlcTask Outputs/MAIN.InMoldDrying.BottomMoldA.HeatingZone[6].qxPWMOut1 <-> Channel 4/Output
//     PlcTask Outputs/MAIN.InMoldDrying.BottomMoldA.HeatingZone[6].qxPWMOut2 <-> Channel 5/Output
//     PlcTask Outputs/MAIN.InMoldDrying.BottomMoldA.HeatingZone[6].qxPWMOut3 <-> Channel 6/Output
//     PlcTask Outputs/MAIN.InMoldDrying.TopMoldB.HeatingZone[1].qxPWMOut1 <-> Channel 8/Output
//     PlcTask Outputs/MAIN.InMoldDrying.TopMoldB.HeatingZone[1].qxPWMOut2 <-> Channel 9/Output
//     PlcTask Outputs/MAIN.InMoldDrying.TopMoldB.HeatingZone[1].qxPWMOut3 <-> Channel 10/Output
//     PlcTask Outputs/MAIN.InMoldDrying.TopMoldB.HeatingZone[2].qxPWMOut1 <-> Channel 11/Output
//     PlcTask Outputs/MAIN.InMoldDrying.TopMoldB.HeatingZone[2].qxPWMOut2 <-> Channel 12/Output
//     PlcTask Outputs/MAIN.InMoldDrying.TopMoldB.HeatingZone[2].qxPWMOut3 <-> Channel 13/Output
//     PlcTask Outputs/MAIN.InMoldDrying.TopMoldB.HeatingZone[3].qxPWMOut1 <-> Channel 14/Output
//     PlcTask Outputs/MAIN.InMoldDrying.TopMoldB.HeatingZone[3].qxPWMOut2 <-> Channel 15/Output
//     PlcTask Outputs/MAIN.InMoldDrying.TopMoldB.HeatingZone[3].qxPWMOut3 <-> Channel 16/Output
//   IMD_PLC/IMD_PLC Instance <-> Device 2 (EtherCAT)/MCC01_600A1 (EK1100)/600A26 (EL2809)
//     PlcTask Outputs/MAIN.InMoldDrying.BottomMoldB.HeatingZone[1].qxPWMOut1 <-> Channel 11/Output
//     PlcTask Outputs/MAIN.InMoldDrying.BottomMoldB.HeatingZone[1].qxPWMOut2 <-> Channel 12/Output
//     PlcTask Outputs/MAIN.InMoldDrying.BottomMoldB.HeatingZone[1].qxPWMOut3 <-> Channel 13/Output
//     PlcTask Outputs/MAIN.InMoldDrying.BottomMoldB.HeatingZone[2].qxPWMOut1 <-> Channel 14/Output
//     PlcTask Outputs/MAIN.InMoldDrying.BottomMoldB.HeatingZone[2].qxPWMOut2 <-> Channel 15/Output
//     PlcTask Outputs/MAIN.InMoldDrying.BottomMoldB.HeatingZone[2].qxPWMOut3 <-> Channel 16/Output
//     PlcTask Outputs/MAIN.InMoldDrying.TopMoldB.HeatingZone[4].qxPWMOut1 <-> Channel 1/Output
//     PlcTask Outputs/MAIN.InMoldDrying.TopMoldB.HeatingZone[4].qxPWMOut2 <-> Channel 2/Output
//     PlcTask Outputs/MAIN.InMoldDrying.TopMoldB.HeatingZone[4].qxPWMOut3 <-> Channel 3/Output
//     PlcTask Outputs/MAIN.InMoldDrying.TopMoldB.HeatingZone[5].qxPWMOut1 <-> Channel 4/Output
//     PlcTask Outputs/MAIN.InMoldDrying.TopMoldB.HeatingZone[5].qxPWMOut2 <-> Channel 5/Output
//     PlcTask Outputs/MAIN.InMoldDrying.TopMoldB.HeatingZone[5].qxPWMOut3 <-> Channel 6/Output
//     PlcTask Outputs/MAIN.InMoldDrying.TopMoldB.HeatingZone[6].qxPWMOut1 <-> Channel 7/Output
//     PlcTask Outputs/MAIN.InMoldDrying.TopMoldB.HeatingZone[6].qxPWMOut2 <-> Channel 8/Output
//     PlcTask Outputs/MAIN.InMoldDrying.TopMoldB.HeatingZone[6].qxPWMOut3 <-> Channel 9/Output
//   IMD_PLC/IMD_PLC Instance <-> Device 2 (EtherCAT)/MCC01_600A1 (EK1100)/600A27 (EL2809)
//     PlcTask Outputs/MAIN.InMoldDrying.BottomMoldB.HeatingZone[3].qxPWMOut1 <-> Channel 1/Output
//     PlcTask Outputs/MAIN.InMoldDrying.BottomMoldB.HeatingZone[3].qxPWMOut2 <-> Channel 2/Output
//     PlcTask Outputs/MAIN.InMoldDrying.BottomMoldB.HeatingZone[3].qxPWMOut3 <-> Channel 3/Output
//     PlcTask Outputs/MAIN.InMoldDrying.BottomMoldB.HeatingZone[4].qxPWMOut1 <-> Channel 4/Output
//     PlcTask Outputs/MAIN.InMoldDrying.BottomMoldB.HeatingZone[4].qxPWMOut2 <-> Channel 5/Output
//     PlcTask Outputs/MAIN.InMoldDrying.BottomMoldB.HeatingZone[4].qxPWMOut3 <-> Channel 6/Output
//     PlcTask Outputs/MAIN.InMoldDrying.BottomMoldB.HeatingZone[5].qxPWMOut1 <-> Channel 7/Output
//     PlcTask Outputs/MAIN.InMoldDrying.BottomMoldB.HeatingZone[5].qxPWMOut2 <-> Channel 8/Output
//     PlcTask Outputs/MAIN.InMoldDrying.BottomMoldB.HeatingZone[5].qxPWMOut3 <-> Channel 9/Output
//     PlcTask Outputs/MAIN.InMoldDrying.BottomMoldB.HeatingZone[6].qxPWMOut1 <-> Channel 10/Output
//     PlcTask Outputs/MAIN.InMoldDrying.BottomMoldB.HeatingZone[6].qxPWMOut2 <-> Channel 11/Output
//     PlcTask Outputs/MAIN.InMoldDrying.BottomMoldB.HeatingZone[6].qxPWMOut3 <-> Channel 12/Output
//   IMD_PLC/IMD_PLC Instance <-> Device 2 (EtherCAT)/MCC01_600A1 (EK1100)/600A4_TwinsafeController (EL6900)
//     PlcTask Inputs/MAIN.ComErr <-> StandardInputs/Standard Out Var 211
//     PlcTask Inputs/MAIN.FbError <-> StandardInputs/Standard Out Var 210
//     PlcTask Inputs/MAIN.OutErr <-> StandardInputs/Standard Out Var 212
//     PlcTask Inputs/MAIN.ixTwinSafe_SafetyRelay[{1..7}] <-> StandardInputs/Standard Out Var {201..207}  (7 links)
//     PlcTask Outputs/MAIN.qxTwinSafe_Reset <-> StandardOutputs/Standard In Var 1
//   IMD_PLC/IMD_PLC Instance <-> Device 2 (EtherCAT)/MCC02_600A1 (EK1100)/MCC02_600A2 (EL1904)
//     PlcTask Inputs/MAIN.InMoldDrying.TopMoldA.HydraulicCilinder.ixEndSwitchA <-> Module 1 (FSOES)/TxPDO/FSOE/InputChannel1
//     PlcTask Inputs/MAIN.InMoldDrying.TopMoldA.HydraulicCilinder.ixEndSwitchB <-> Module 1 (FSOES)/TxPDO/FSOE/InputChannel2
//     PlcTask Inputs/MAIN.InMoldDrying.TransferMold.HydraulicCilinder.ixEndSwitchA <-> Module 1 (FSOES)/TxPDO/FSOE/InputChannel3
//     PlcTask Inputs/MAIN.InMoldDrying.TransferMold.HydraulicCilinder.ixEndSwitchB <-> Module 1 (FSOES)/TxPDO/FSOE/InputChannel4
//   IMD_PLC/IMD_PLC Instance <-> Device 2 (EtherCAT)/MCC02_600A1 (EK1100)/MCC02_600A3 (EL1904)
//     PlcTask Inputs/MAIN.InMoldDrying.TopMoldB.HydraulicCilinder.ixEndSwitchA <-> Module 1 (FSOES)/TxPDO/FSOE/InputChannel1
//     PlcTask Inputs/MAIN.InMoldDrying.TopMoldB.HydraulicCilinder.ixEndSwitchB <-> Module 1 (FSOES)/TxPDO/FSOE/InputChannel2
//   IMD_PLC/IMD_PLC Instance <-> Device 2 (EtherCAT)/MCC02_600A1 (EK1100)/MCC02_600A5 (EL1809)
//     PlcTask Inputs/MAIN.InMoldDrying.HydraulicsMain.CoolingFan.ixMaintenance <-> Channel 15/Input
//     PlcTask Inputs/MAIN.InMoldDrying.HydraulicsMain.CoolingFan.ixRunning <-> Channel 14/Input
//     PlcTask Inputs/MAIN.InMoldDrying.HydraulicsMain.CoolingFan.ixThermal <-> Channel 13/Input
//     PlcTask Inputs/MAIN.InMoldDrying.HydraulicsMain.FilterMotor.ixMaintenance <-> Channel 12/Input
//     PlcTask Inputs/MAIN.InMoldDrying.HydraulicsMain.FilterMotor.ixRunning <-> Channel 11/Input
//     PlcTask Inputs/MAIN.InMoldDrying.HydraulicsMain.FilterMotor.ixThermal <-> Channel 10/Input
//     PlcTask Inputs/MAIN.InMoldDrying.HydraulicsMain.HydraulicPump.ixIsRunning <-> Channel 6/Input
//     PlcTask Inputs/MAIN.InMoldDrying.HydraulicsMain.HydraulicPump.ixMaintenance <-> Channel 9/Input
//     PlcTask Inputs/MAIN.InMoldDrying.HydraulicsMain.HydraulicPump.ixSSFailure <-> Channel 7/Input
//     PlcTask Inputs/MAIN.InMoldDrying.HydraulicsMain.ixCabinetCoolerError <-> Channel 2/Input
//     PlcTask Inputs/MAIN.InMoldDrying.HydraulicsMain.ixHydraulicsMcc24vError <-> Channel 1/Input
//   IMD_PLC/IMD_PLC Instance <-> Device 2 (EtherCAT)/MCC02_600A1 (EK1100)/MCC02_600A6 (EL1809)
//     PlcTask Inputs/MAIN.InMoldDrying.HydraulicsMain.ixAuxFilterAt100 <-> Channel 7/Input
//     PlcTask Inputs/MAIN.InMoldDrying.HydraulicsMain.ixAuxFilterAt75 <-> Channel 6/Input
//     PlcTask Inputs/MAIN.InMoldDrying.HydraulicsMain.ixOilLvlLow <-> Channel 9/Input
//     PlcTask Inputs/MAIN.InMoldDrying.HydraulicsMain.ixOilLvlTooLow <-> Channel 8/Input
//     PlcTask Inputs/MAIN.InMoldDrying.HydraulicsMain.ixPressureFilterAt100 <-> Channel 5/Input
//     PlcTask Inputs/MAIN.InMoldDrying.HydraulicsMain.ixPressureFilterAt75 <-> Channel 4/Input
//     PlcTask Inputs/MAIN.InMoldDrying.HydraulicsMain.ixTemperatureSwitch40c <-> Channel 10/Input
//     PlcTask Inputs/MAIN.InMoldDrying.HydraulicsMain.ixTemperatureSwitch55c <-> Channel 11/Input
//     PlcTask Inputs/MAIN.InMoldDrying.HydraulicsMain.ixTemperatureSwitchTooHigh <-> Channel 12/Input
//     PlcTask Inputs/MAIN.InMoldDrying.TopMoldA.HydraulicCilinder.ixMSPAReadyToOperate <-> Channel 1/Input
//     PlcTask Inputs/MAIN.InMoldDrying.TopMoldB.HydraulicCilinder.ixMSPAReadyToOperate <-> Channel 3/Input
//     PlcTask Inputs/MAIN.InMoldDrying.TransferMold.HydraulicCilinder.ixMSPAReadyToOperate <-> Channel 2/Input
//   IMD_PLC/IMD_PLC Instance <-> Device 2 (EtherCAT)/MCC02_600A1 (EK1100)/MCC02_600A8 (EL2809)
//     PlcTask Outputs/MAIN.InMoldDrying.HydraulicsMain.CoolingFan.Q <-> Channel 3/Output
//     PlcTask Outputs/MAIN.InMoldDrying.HydraulicsMain.FilterMotor.Q <-> Channel 2/Output
//     PlcTask Outputs/MAIN.InMoldDrying.HydraulicsMain.HydraulicPump.Q <-> Channel 1/Output
//     PlcTask Outputs/MAIN.InMoldDrying.HydraulicsMain.IsolationValve.Q <-> Channel 10/Output
//     PlcTask Outputs/MAIN.InMoldDrying.HydraulicsMain.PressurizePumpValve.Q <-> Channel 9/Output
//     PlcTask Outputs/MAIN.InMoldDrying.TopMoldA.HydraulicCilinder.qxMSPAEnable <-> Channel 5/Output
//     PlcTask Outputs/MAIN.InMoldDrying.TopMoldB.HydraulicCilinder.qxMSPAEnable <-> Channel 7/Output
//     PlcTask Outputs/MAIN.InMoldDrying.TransferMold.HydraulicCilinder.qxMSPAEnable <-> Channel 6/Output
//   IMD_PLC/IMD_PLC Instance <-> Device 2 (EtherCAT)/MCC02_600A1 (EK1100)/MCC02_600A9 (EL4134)
//     PlcTask Outputs/MAIN.InMoldDrying.TopMoldA.HydraulicCilinder.HydraulicValve.qwOutput <-> AO Output Channel 1/Analog output
//     PlcTask Outputs/MAIN.InMoldDrying.TopMoldB.HydraulicCilinder.HydraulicValve.qwOutput <-> AO Output Channel 2/Analog output
//     PlcTask Outputs/MAIN.InMoldDrying.TransferMold.HydraulicCilinder.HydraulicValve.qwOutput <-> AO Output Channel 3/Analog output
//   IMD_PLC/IMD_PLC Instance <-> NC-Task 1 SAF/Axes/BottomMoldA
//     PlcTask Inputs/MAIN.InMoldDrying.BottomMoldA.HorizontalAxis.axAxis.NcToPlc <-> Outputs/ToPlc
//     PlcTask Outputs/MAIN.InMoldDrying.BottomMoldA.HorizontalAxis.axAxis.PlcToNc <-> Inputs/FromPlc
//   IMD_PLC/IMD_PLC Instance <-> NC-Task 1 SAF/Axes/BottomMoldB
//     PlcTask Inputs/MAIN.InMoldDrying.BottomMoldB.HorizontalAxis.axAxis.NcToPlc <-> Outputs/ToPlc
//     PlcTask Outputs/MAIN.InMoldDrying.BottomMoldB.HorizontalAxis.axAxis.PlcToNc <-> Inputs/FromPlc
//   IMD_PLC/IMD_PLC Instance <-> NC-Task 1 SAF/Axes/GantryA_Hor
//     PlcTask Inputs/MAIN.ProductHandling.GantryA.HorizontalAxis.axAxis.NcToPlc <-> Outputs/ToPlc
//     PlcTask Outputs/MAIN.ProductHandling.GantryA.HorizontalAxis.axAxis.PlcToNc <-> Inputs/FromPlc
//   IMD_PLC/IMD_PLC Instance <-> NC-Task 1 SAF/Axes/GantryA_Ver
//     PlcTask Inputs/MAIN.ProductHandling.GantryA.VerticalAxis.axAxis.NcToPlc <-> Outputs/ToPlc
//     PlcTask Outputs/MAIN.ProductHandling.GantryA.VerticalAxis.axAxis.PlcToNc <-> Inputs/FromPlc
//   IMD_PLC/IMD_PLC Instance <-> NC-Task 1 SAF/Axes/GantryB_Hor
//     PlcTask Inputs/MAIN.ProductHandling.GantryB.HorizontalAxis.axAxis.NcToPlc <-> Outputs/ToPlc
//     PlcTask Outputs/MAIN.ProductHandling.GantryB.HorizontalAxis.axAxis.PlcToNc <-> Inputs/FromPlc
//   IMD_PLC/IMD_PLC Instance <-> NC-Task 1 SAF/Axes/GantryB_Ver
//     PlcTask Inputs/MAIN.ProductHandling.GantryB.VerticalAxis.axAxis.NcToPlc <-> Outputs/ToPlc
//     PlcTask Outputs/MAIN.ProductHandling.GantryB.VerticalAxis.axAxis.PlcToNc <-> Inputs/FromPlc
//   IMD_PLC/IMD_PLC Instance <-> NC-Task 1 SAF/Axes/SprayBar
//     PlcTask Inputs/MAIN.InMoldDrying.ProductForming.SprayBarMotor.axAxis.NcToPlc <-> Outputs/ToPlc
//     PlcTask Outputs/MAIN.InMoldDrying.ProductForming.SprayBarMotor.axAxis.PlcToNc <-> Inputs/FromPlc
//   IMD_PLC/IMD_PLC Instance <-> SpeedControl/SpeedControl Instance
//     PlcTask Inputs/MAIN.ComSC.SpeedControl_IMD <-> PlcTask_SpeedControl Outputs/MAIN.ComSpeedControl_IMD1.SpeedControl_IMD
//     PlcTask Outputs/MAIN.ComSC.IMD_SpeedControl <-> PlcTask_SpeedControl Inputs/MAIN.ComSpeedControl_IMD1.IMD_SpeedControl
//   SpeedControl/SpeedControl Instance <-> Device 2 (EtherCAT)/MCC01_2_610A1 (EK1100)/610A2 (EK1122)/Drive A-Belt / B-Spraybar (AX5201-0000-0203)
//     PlcTask_SpeedControl Inputs/MAIN.Conveyor.Belt.iDriveRef/aNetId <-> InfoData/AdsAddr/netId
//     PlcTask_SpeedControl Inputs/MAIN.Conveyor.Belt.iDriveRef/nDriveNo <-> InfoData/Chn0
//     PlcTask_SpeedControl Inputs/MAIN.Conveyor.Belt.iDriveRef/nSlaveAddr <-> InfoData/AdsAddr/port
//   SpeedControl/SpeedControl Instance <-> Device 2 (EtherCAT)/MCC01_2_610A1 (EK1100)/610A2 (EK1122)/EJBox (EP9128-0021)/EPP_SensorSpeedControl (EPP1322-0001)/Box SpeedControl (EPP6228-0022)
//     PlcTask_SpeedControl Inputs/MAIN.Conveyor.IMD1_GantryB.miSensorPitchClear <-> Module 11 (Digital Inputs)/Digital Inputs/Pin2 Ch1
//   SpeedControl/SpeedControl Instance <-> NC-Task 1 SAF/Axes/Conveyor
//     PlcTask_SpeedControl Inputs/MAIN.Conveyor.Belt.axAxis.NcToPlc <-> Outputs/ToPlc
//     PlcTask_SpeedControl Outputs/MAIN.Conveyor.Belt.axAxis.PlcToNc <-> Inputs/FromPlc

CONFIGURATION IMD_PLC
    RESOURCE PLC ON TwinCAT3
        TASK PlcTask(INTERVAL := T#10ms, PRIORITY := 20);
        PROGRAM MAIN WITH PlcTask : MAIN;
    END_RESOURCE
END_CONFIGURATION

// ---- DUTs/ST_COM_SpeedControl.TcDUT
TYPE ST_COM_SpeedControl :
STRUCT
	IMD_SpeedControl AT %Q*: ST_COM_IMD_SpdCntrl;
	SpeedControl_IMD AT %I*: ST_COM_SpdCntrl_IMD;
END_STRUCT
END_TYPE

// ---- DUTs/ST_COM_IMD_SpdCntrl.TcDUT
TYPE ST_COM_IMD_SpdCntrl :
STRUCT
	Stopped				: BOOL;					// IMD is in stopped state
	RTO					: BOOL;					// IMD is Ready to Operate state			
	BlowOffProcessedA	: ARRAY[1..4] OF BOOL;	// signal to confirm that the blowoff has actually happend for A side
	BlowOffProcessedB	: ARRAY[1..4] OF BOOL;	// signal to confirm that the blowoff has actually happend for B side
	FormingReadyA		: BOOL;					// signal to confirm that the forming has actually started for A side
	FormingReadyB		: BOOL;					// signal to confirm that the forming has actually started for B side	
	GantryA_Ready		: BOOL; 				// signal that Gantry A is in position above the conveyor and ready to blow off
	GantryB_Ready		: BOOL; 				// signal that Gantry B is in position above the conveyor and ready to blow off
	ES					: BOOL;					// Emergency stop from the IMD that also need to stop the conveyor
	MaximumSpeed		: REAL;					// theoretical maximum speed with current settings
	ActualSpeed			: REAL;					// Number of KO's in last cycle
	HMI_Reset			: BOOL;					// MZE 20190311 For testing at LoodsLanghout
END_STRUCT
END_TYPE

// ---- DUTs/ST_MachPar.TcDUT
TYPE ST_MachPar :
STRUCT
	InMoldDrying					: ST_IMDMachPar;
	ProductHandling					: ST_ProductHandlingMachPar;
END_STRUCT
END_TYPE

// ---- DUTs/ST_OEE.TcDUT
TYPE ST_OEE :
STRUCT
	TotalRunTime					: DINT;
	TotalWaitTime					: DINT;
	TotalDownTime					: DINT;
	
	KickOffsAside					: REAL;
	ProducedSheetsASide				: DINT;
	ProducedProductsAside			: DINT;
	
	KickOffsBSide					: REAL;
	ProducedSheetsBSide				: DINT;
	ProducedProductsBside			: DINT;
	
	TotalProducedSheets				: DINT;
	TotalProducedProducts			: DINT;
	KickOffsBothSides				: REAL;
	
	ImdErrorTime					: DINT;
	ProductHandingErrorTime			: DINT;
	
	// Power stuff
	
	// Voltage
	L1_Voltage						: REAL;
	L2_Voltage						: REAL;
	L3_Voltage						: REAL;
	L123_VoltageAverage				: REAL;
	
	// Current
	L1_Current						: REAL;
	L2_Current						: REAL;
	L3_Current						: REAL;
	L123_CurrentAverage				: REAL;
	
	// Power
	L1_Watt							: REAL;
	L2_Watt							: REAL;
	L3_Watt							: REAL;
	L123_WattAverage				: REAL;	
	
	
END_STRUCT
END_TYPE

// ---- DUTs/ST_PowerMeasurement.TcDUT
TYPE ST_PowerMeasurement :
STRUCT
	ixPDOToggle		:BOOL;
	iwCurrent 		:DINT;
	iwVoltage		:DINT;
	iwActivePower	:DINT;
	iwIndex			:USINT;
	iwVariantValue	:DINT;
END_STRUCT
END_TYPE

// ---- DUTs/ST_ProdPar.TcDUT
TYPE ST_ProdPar :
STRUCT
	InMoldDrying			: ST_IMDProdPar;
	ProductHandling			: ST_ProductHandlingProdPar;

END_STRUCT
END_TYPE

